// TwinCAT 3 PLC project TcoCognexVision
// Title: TcoCognexVision
// Company: Vortex.Library
// ProjectVersion: 0.6.0.913
// ProgramVersion: 3.1.4023.0
// libraries:
//   Tc2_Standard, * (Beckhoff Automation GmbH)
//   Tc2_System, * (Beckhoff Automation GmbH)
//   Tc3_Module, * (Beckhoff Automation GmbH)
//   TcoAbstractions, 0.6.0.913 (Vortex.Library)
//   TcoCore, 0.6.0.913 (Vortex.Library)
//   TcoIo, 0.6.0.913 (Vortex.Library)
//   TcoUtilities, 0.6.0.913 (Vortex.Library)
// project tree:
//   / PlcTask.TcTTO (not stored)
//   POUs/TcoDataman/v_5_x_x/IO/ TcoDatamanAcquisitionControl_v_5_x_x.TcDUT (not stored), TcoDatamanAcquisitionStatus_v_5_x_x.TcDUT (not stored), TcoDatamanIO_v_5_x_x.TcDUT (not stored), TcoDatamanResultData_v_5_x_x.TcDUT (not stored), TcoDatamanResultsControl_v_5_x_x.TcDUT (not stored), TcoDatamanResultsStatus_v_5_x_x.TcDUT (not stored), TcoDatamanSoftEventControl_v_5_x_x.TcDUT (not stored), TcoDatamanUserData_v_5_x_x.TcDUT (not stored)
//   POUs/TcoDataman/v_5_x_x/Structs/ eDatamanResultDataSize_v_5_x_x.TcDUT (not stored), eDatamanUserDataSize_v_5_x_x.TcDUT (not stored), TcoDatamanConfig_v_5_x_x.TcDUT, TcoDatamanResults_v_5_x_x.TcDUT (not stored), TcoDatamanSignalStates_v_5_x_x.TcDUT (not stored), TcoDatamanStatus_v_5_x_x.TcDUT, TcoDatamanUser_v_5_x_x.TcDUT (not stored)
//   POUs/TcoDataman/v_5_x_x/Tasks/ TcoDatamanClearResultData_v_5_x_x.TcPOU, TcoDatamanRead_v_5_x_x.TcPOU
//   POUs/TcoDataman/v_5_x_x/ TcoDataman_v_5_x_x.TcPOU
//   POUs/TcoDesigner/Structs/ eTcoDesignerTriggerType.TcDUT (not stored), TcoDesignerConfig_v_2_x_x.TcDUT, TcoDesignerData_2_x_x.TcDUT (not stored), TcoDesignerRootContainer.TcPOU (not stored), TcoDesignerStatus_v_2_x_x.TcDUT (not stored), TcoDesignerGenericResults_v_2_x_x.TcDUT (not stored), TcoDesignerPcToPlc_v_2_x_x.TcDUT (not stored), TcoDesignerPlcToPc_v_2_x_x.TcDUT (not stored)
//   POUs/TcoDesigner/Tasks/ TcoDesignerTrigger_v_2_x_x.TcPOU, TcoDesignerClearInspectionResults_v_2_x_x.TcPOU
//   POUs/TcoDesigner/ TcoDesigner_v_2_x_x.TcPOU (not stored)
//   POUs/TcoInsight/v_5_x_x/IO/ TcoInsightAcquisitionControl_v_5_x_x.TcDUT (not stored), TcoInsightAcquisitionStatus_v_5_x_x.TcDUT (not stored), TcoInsightIO_v_5_x_x.TcDUT (not stored), TcoInsightResultData_v_5_x_x.TcDUT (not stored), TcoInsightInspectionControl_v_5_x_x.TcDUT (not stored), TcoInsightInspectionStatus_v_5_x_x.TcDUT (not stored), TcoInsightSoftEventControl_v_5_x_x.TcDUT (not stored), TcoInsightCommandControl_v_5_x_x.TcDUT (not stored), TcoInsightUserData_v_5_x_x.TcDUT (not stored)
//   POUs/TcoInsight/v_5_x_x/Structs/ eTcoInsightResultDataSize_v_5_x_x.TcDUT (not stored), eTcoInsightUserDataSize_v_5_x_x.TcDUT (not stored), TcoInsightConfig_v_5_x_x.TcDUT, TcoInsightResults_v_5_x_x.TcDUT (not stored), TcoInsightSignalStates_v_5_x_x.TcDUT (not stored), TcoInsightStatus_v_5_x_x.TcDUT (not stored), TcoInsightUser_v_5_x_x.TcDUT (not stored)
//   POUs/TcoInsight/v_5_x_x/Tasks/ TcoInsightSetUserData_v_5_x_x.TcPOU, TcoInsightClearUserData_v_5_x_x.TcPOU, TcoInsightTrigger_v_5_x_x.TcPOU, TcoInsightChangeJobByName_v_5_x_x.TcPOU, TcoInsightChangeJobByNumber_v_5_x_x.TcPOU, TcoInsightClearInspectionResults_v_5_x_x.TcPOU, TcoInsightSoftEvent_v_5_x_x.TcPOU
//   POUs/TcoInsight/v_5_x_x/ TcoInsight_v_5_x_x.TcPOU
//   POUs/ TcoVisionParams.TcGVL (not stored)

// ---- POUs/TcoDataman/v_5_x_x/Structs/TcoDatamanConfig_v_5_x_x.TcDUT
TYPE
    TcoDatamanConfig_v_5_x_x :
    STRUCT
        ResultDataSize : eDatamanResultDataSize_v_5_x_x := eDatamanResultDataSize_v_5_x_x.RESULT_DATA_64B;
        UserDataSize : eDatamanUserDataSize_v_5_x_x := eDatamanUserDataSize_v_5_x_x.USER_DATA_64B;
        DataFormat : eTcoDataFormat := TcoUtilities.eTcoDataFormat.BigEndian;
		{attribute addProperty Name "<#Continuous Reading (Hand-held reader)#>"}
        ContinuousReading : BOOL := FALSE;
		UpdateStatesPermanently : BOOL := TRUE;
        InfoTime : TIME := T#2S;
        ErrorTime : TIME := T#5S;
		ShowUserData : BOOL := FALSE;
		ShowResultsData : BOOL := FALSE;
    END_STRUCT
END_TYPE

// ---- POUs/TcoDataman/v_5_x_x/Structs/TcoDatamanStatus_v_5_x_x.TcDUT
TYPE TcoDatamanStatus_v_5_x_x :
STRUCT
	ActionDescription : STRING(100);
	ResultString:STRING(254);
	
	SignalStatus : TcoDatamanSignalStates_v_5_x_x;
END_STRUCT
END_TYPE

// ---- POUs/TcoDesigner/Structs/TcoDesignerConfig_v_2_x_x.TcDUT
TYPE
    TcoDesignerConfig_v_2_x_x :
    STRUCT
   
      
		TriggerTimemout : TIME := T#15S;
		ConnectionTimemout : TIME := T#10S;
        InfoTime : TIME := T#2S;
        ErrorTime : TIME := T#0S;
    END_STRUCT
END_TYPE

// ---- POUs/TcoInsight/v_5_x_x/Structs/TcoInsightConfig_v_5_x_x.TcDUT
TYPE
    TcoInsightConfig_v_5_x_x :
    STRUCT
        ResultDataSize : eTcoInsightResultDataSize_v_5_x_x := eTcoInsightResultDataSize_v_5_x_x.RESULT_DATA_64B;
        UserDataSize : eTcoInsightUserDataSize_v_5_x_x := eTcoInsightUserDataSize_v_5_x_x.USER_DATA_64B;
        DataFormat : eTcoDataFormat := TcoUtilities.eTcoDataFormat.BigEndian;
		UpdateStatesPermanently : BOOL := FALSE;
        MaxJobNumber : UINT := 999;
        InfoTime : TIME := T#2S;
        ErrorTime : TIME := T#0S;
		ShowUserData : BOOL := FALSE;
		ShowResultsData : BOOL := FALSE;

    //	ServiceJobNumber		:	UINT;
    //	ServiceJobName			:	STRING;
    //	ServiceSoftEventNumber	:	UINT;
    END_STRUCT
END_TYPE

// ---- POUs/TcoDataman/v_5_x_x/Tasks/TcoDatamanClearResultData_v_5_x_x.TcPOU
FUNCTION_BLOCK TcoDatamanClearResultData_v_5_x_x EXTENDS TcoCore.TcoTask
VAR_IN_OUT
	inoIoData : TcoDatamanIO_v_5_x_x;
    inoConfig : TcoDatamanConfig_v_5_x_x;
	inoStatus : TcoDatamanStatus_v_5_x_x;	
	inoResults : TcoDatamanResults_v_5_x_x;
END_VAR
VAR
    {attribute 'hide'} 
	_progress : INT := 0;
    {attribute 'hide'} 
	_infoTimer :  TON;
    {attribute 'hide'} 
	_errorTimer :  TON;
    {attribute 'hide'} 
	_varInfo : __SYSTEM.VAR_INFO;
    {attribute 'hide'} 
	_sb : TcoCore.StringBuilder;
END_VAR

IF Execute() THEN
	IF _progress = 0 THEN
		IF NOT __ISVALIDREF(inoIoData) THEN
			_varInfo :=__VARINFO(inoIoData);
			Messenger.Programming(_sb.Clear().Append('<#Invalid reference: #>').Append(_varInfo.Symbol).ToString()).Pin();
		ELSIF NOT __ISVALIDREF(inoConfig) THEN                                                  
			_varInfo :=__VARINFO(inoConfig);                                                    
			Messenger.Programming(_sb.Clear().Append('<#Invalid reference: #>').Append(_varInfo.Symbol).ToString()).Pin();
		ELSIF NOT __ISVALIDREF(inoStatus) THEN                                                  
			_varInfo :=__VARINFO(inoStatus);                                                    
			Messenger.Programming(_sb.Clear().Append('<#Invalid reference: #>').Append(_varInfo.Symbol).ToString()).Pin();
		ELSIF NOT __ISVALIDREF(inoResults) THEN                                              
			_varInfo :=__VARINFO(inoResults);                                                
			Messenger.Programming(_sb.Clear().Append('<#Invalid reference: #>').Append(_varInfo.Symbol).ToString()).Pin();
		ELSE
			_progress := _progress + 1;
		END_IF
	END_IF
	
	IF _progress = 1 THEN
		THIS^.inoStatus.ActionDescription := '<#Clearing of the result data running.#>'; 
		CallTimers(FALSE);
		_progress := _progress + 1;
	END_IF
	
	IF _progress = 2 THEN
		THIS^.inoIoData.AcquisitionControl.TriggerEnable := FALSE;
		THIS^.inoIoData.AcquisitionControl.Trigger := FALSE;
		THIS^.inoIoData.ResultsControl.ResultsAcknowledge := TRUE;
		THIS^.Messenger.OnCondition(_infoTimer.Q).Warning('<#Waiting for the result data cleared!#>').Pin();
		THIS^.inoResults.Length := 0; 
		IF Tc2_System.MEMSET(destAddr:= ADR(THIS^.inoResults.Data) , fillByte:= 0 , n:= SIZEOF(THIS^.inoResults.Data)) >0 THEN
			CallTimers(FALSE);
			_progress := _progress + 1;
		END_IF
	END_IF
	
	IF _progress = 3 THEN
		THIS^.Messenger.OnCondition(_infoTimer.Q).Warning('<#Waiting for the signal ResultsAvailable to be reseted!#>').Pin(); 
		IF NOT THIS^.inoIoData.ResultsStatus.ResultsAvailable THEN
			CallTimers(FALSE);
			_progress := _progress + 1;
		END_IF
	END_IF
	
	IF _progress = 4 THEN
		THIS^.inoIoData.ResultsControl.ResultsAcknowledge := FALSE;
		THIS^.DoneWhen(TRUE);
		CallTimers(FALSE);
		_progress := 0;
	END_IF
	
	CallTimers(TRUE);
	
	THIS^.ThrowWhen(_errorTimer.Q);
END_IF

METHOD CallTimers
VAR_INPUT
	inValue : BOOL;
END_VAR
IF  __ISVALIDREF(inoConfig) AND THIS^.inoConfig.ErrorTime <> T#0S OR NOT inValue THEN  
_errorTimer(IN := inValue, PT := THIS^.inoConfig.ErrorTime);
END_IF;
IF  __ISVALIDREF(inoConfig) AND THIS^.inoConfig.InfoTime <>T#0S OR NOT inValue THEN  
_infoTimer(IN := inValue, PT := THIS^.inoConfig.InfoTime);
END_IF;
END_METHOD

{attribute 'hide'}
METHOD PUBLIC FB_init : BOOL
VAR_INPUT
	bInitRetains : BOOL; // if TRUE, the retain variables are initialized (warm start / cold start)
	bInCopyCode : BOOL;  // if TRUE, the instance afterwards gets moved into the copy code (online change)
	ParentObject : ITcoObject;
END_VAR
END_METHOD

(*~
	<docu>
		<summary>
			Executes when task is aborted.
		</summary>			
	</docu>	
~*)
METHOD PROTECTED OnAbort
THIS^.inoStatus.ActionDescription := '<#Clearing of the result data was aborted, while not yet completed!#>';
END_METHOD

(*~
	<docu>
		<summary>
			Executes when task reaches the ```Done``` state .
		</summary>			
	</docu>	
~*)
METHOD PROTECTED OnDone
THIS^.inoStatus.ActionDescription := '<#Clearing of the result data was completed successfully.#>';
END_METHOD

(*~
	<docu>
		<summary>
			Executes when task reaches the ```Error``` state.
			<para>
				Do not confuse with <see cref="PlcDocu.TcoCore.TcoTask.WhileError()"/>, that is called cyclically until '''Error''' state is left.
			</para>
		</summary>			
	</docu>	
~*)
METHOD PROTECTED OnError
THIS^.inoStatus.ActionDescription := '<#Clearing of the result data finished with error.#>';
END_METHOD

METHOD PROTECTED OnStart
THIS^.inoStatus.ActionDescription := '<#Clearing of the result data started.#>';
END_METHOD

(*~
	<docu>
		<summary>
			Restores this instance to the Ready state. Can be called explicitly or from within one of the restore mechanisms.
			<para>
				See also <see cref="PlcDocu.TcoCore.TcoTask.AutoRestorable()"/>
			</para>
		</summary>			
	</docu>	
~*)
METHOD Restore : ITcoRestorable
SUPER^.Restore();
_progress := 0;
CallTimers(FALSE);
Messenger.UnPin();
END_METHOD

END_FUNCTION_BLOCK

// ---- POUs/TcoDataman/v_5_x_x/Tasks/TcoDatamanRead_v_5_x_x.TcPOU
FUNCTION_BLOCK TcoDatamanRead_v_5_x_x EXTENDS TcoCore.TcoTask
VAR_IN_OUT
	inoIoData 	: TcoDatamanIO_v_5_x_x;
    inoConfig 	: TcoDatamanConfig_v_5_x_x;
	inoStatus 	: TcoDatamanStatus_v_5_x_x;	
	inoResults 	: TcoDatamanResults_v_5_x_x;
END_VAR
VAR
    {attribute 'hide'} 
	_progress : INT := 0;
    {attribute 'hide'} 
	_infoTimer :  TON;
    {attribute 'hide'} 
	_errorTimer :  TON;
    {attribute 'hide'} 
	_varInfo : __SYSTEM.VAR_INFO;
    {attribute 'hide'} 
	_sb : TcoCore.StringBuilder;
END_VAR

IF Execute() THEN
	IF _progress = 0 THEN
		IF NOT __ISVALIDREF(inoIoData) THEN
			_varInfo :=__VARINFO(inoIoData);
			Messenger.Programming(_sb.Clear().Append('<#Invalid reference: #>').Append(_varInfo.Symbol).ToString()).Pin();
		ELSIF NOT __ISVALIDREF(inoConfig) THEN                                                  
			_varInfo :=__VARINFO(inoConfig);                                                    
			Messenger.Programming(_sb.Clear().Append('<#Invalid reference: #>').Append(_varInfo.Symbol).ToString()).Pin();
		ELSIF NOT __ISVALIDREF(inoStatus) THEN                                                  
			_varInfo :=__VARINFO(inoStatus);                                                    
			Messenger.Programming(_sb.Clear().Append('<#Invalid reference: #>').Append(_varInfo.Symbol).ToString()).Pin();
		ELSIF NOT __ISVALIDREF(inoResults) THEN                                              
			_varInfo :=__VARINFO(inoResults);                                                
			Messenger.Programming(_sb.Clear().Append('<#Invalid reference: #>').Append(_varInfo.Symbol).ToString()).Pin();
		ELSE
			_progress := _progress + 1;
		END_IF
	END_IF
	
	IF _progress = 1 THEN
		THIS^.inoStatus.ActionDescription := '<#Reading running.#>'; 
		CallTimers(FALSE);
		_progress := _progress + 1;
	END_IF
	
	IF _progress = 2 THEN
		THIS^.inoIoData.AcquisitionControl.TriggerEnable := TRUE;
		THIS^.inoIoData.AcquisitionControl.Trigger := FALSE;
		THIS^.inoIoData.ResultsControl.EnableResultBuffering := FALSE;
		THIS^.inoIoData.ResultsControl.ResultsAcknowledge := THIS^.inoIoData.ResultsStatus.ResultsAvailable;
		THIS^.Messenger.OnCondition(_infoTimer.Q).Warning('<#Waiting for the signal ResultsAvailable to be reseted!#>').Pin(); 
		IF NOT THIS^.inoIoData.ResultsStatus.ResultsAvailable THEN
			CallTimers(FALSE);
			_progress := _progress + 1;
		END_IF
	END_IF
	
	IF _progress = 3 THEN
		THIS^.Messenger.OnCondition(_infoTimer.Q).Warning('<#Waiting for the signal TriggerReady to be set!#>').Pin(); 
		IF THIS^.inoIoData.AcquisitionStatus.TriggerReady THEN
			CallTimers(FALSE);
			_progress := _progress + 1;
		END_IF
	END_IF
	
	IF _progress = 4 THEN
		THIS^.inoIoData.AcquisitionControl.Trigger := TRUE;
		THIS^.Messenger.OnCondition(_infoTimer.Q).Warning('<#Waiting for the signal TriggerAcknowledge to be set!#>').Pin(); 
		IF THIS^.inoIoData.AcquisitionStatus.TriggerAcknowledge THEN
			CallTimers(FALSE);
			_progress := _progress + 1;
		END_IF
	END_IF
	
	IF _progress = 5 THEN
		THIS^.Messenger.OnCondition(_infoTimer.Q).Warning('<#Waiting for the signal ResultsAvailable to be set!#>').Pin(); 
		IF THIS^.inoIoData.ResultsStatus.ResultsAvailable THEN
			CallTimers(FALSE);
			_progress := _progress + 1;
		END_IF
	END_IF
	
	IF _progress = 6 THEN
		THIS^.inoResults.Length := THIS^.inoIoData.ResultData.ResultLength;
		THIS^.Messenger.OnCondition(_infoTimer.Q).Warning('<#Waiting for the ResultData copied!#>').Pin(); 
		IF  THIS^.inoIoData.ResultData.ResultCode.0=1 THEN // read successfull
			IF Tc2_System.MEMCPY(srcAddr := ADR(THIS^.inoIoData.ResultData.ResultData) , destAddr:= ADR(THIS^.inoResults.Data) ,  n:= THIS^.inoResults.Length) > 0 AND 
				Tc2_System.MEMSET(destAddr:= ADR(THIS^.inoResults.Data) + THIS^.inoResults.Length, fillByte:= 0 , n:= SIZEOF(THIS^.inoResults.Data) - THIS^.inoResults.Length)>0 THEN
				CallTimers(FALSE);
				_progress := _progress + 1;
			END_IF;
		ELSIF THIS^.inoIoData.ResultData.ResultCode.0=0  THEN  // read not successfull
			Tc2_System.MEMSET(destAddr:= ADR(THIS^.inoIoData) , fillByte:= 0 , n:= SIZEOF(THIS^.inoIoData));
			CallTimers(FALSE);
			_progress := _progress + 1;
		
		END_IF
	END_IF
	
	IF _progress = 7 THEN
		THIS^.inoIoData.AcquisitionControl.Trigger := FALSE;
		THIS^.inoIoData.ResultsControl.EnableResultBuffering := FALSE;
		THIS^.inoIoData.ResultsControl.ResultsAcknowledge := TRUE;
		//THIS^.ThrowWhen(THIS^.inoIoData.ResultData.ResultCode=0 OR THIS^.inoIoData.ResultData.ResultLength=0);
		THIS^.DoneWhen(TRUE);
		_progress := 0;
	END_IF
	THIS^.ThrowWhen(THIS^.inoIoData.AcquisitionStatus.MissedAcquisition );
	THIS^.ThrowWhen(THIS^.inoIoData.ResultsStatus.ErrorDetected);

	CallTimers(TRUE);
	
	THIS^.ThrowWhen(_errorTimer.Q);
	
END_IF

METHOD CallTimers
VAR_INPUT
	inValue : BOOL;
END_VAR
IF  __ISVALIDREF(inoConfig) AND THIS^.inoConfig.ErrorTime <> T#0S OR NOT inValue THEN  
_errorTimer(IN := inValue, PT := THIS^.inoConfig.ErrorTime);
END_IF;
IF  __ISVALIDREF(inoConfig) AND THIS^.inoConfig.InfoTime <>T#0S OR NOT inValue THEN  
_infoTimer(IN := inValue, PT := THIS^.inoConfig.InfoTime);
END_IF;
END_METHOD

{attribute 'hide'}
METHOD PUBLIC FB_init : BOOL
VAR_INPUT
	bInitRetains : BOOL; // if TRUE, the retain variables are initialized (warm start / cold start)
	bInCopyCode : BOOL;  // if TRUE, the instance afterwards gets moved into the copy code (online change)
	ParentObject : ITcoObject;
END_VAR
END_METHOD

(*~
	<docu>
		<summary>
			Executes when task is aborted.
		</summary>			
	</docu>	
~*)
METHOD PROTECTED OnAbort
THIS^.inoStatus.ActionDescription := '<#Reading was aborted, while not yet completed!#>';
END_METHOD

(*~
	<docu>
		<summary>
			Executes when task reaches the ```Done``` state .
		</summary>			
	</docu>	
~*)
METHOD PROTECTED OnDone
THIS^.inoStatus.ActionDescription := '<#Reading was completed successfully.#>';
END_METHOD

(*~
	<docu>
		<summary>
			Executes when task reaches the ```Error``` state.
			<para>
				Do not confuse with <see cref="PlcDocu.TcoCore.TcoTask.WhileError()"/>, that is called cyclically until '''Error''' state is left.
			</para>
		</summary>			
	</docu>	
~*)
METHOD PROTECTED OnError
THIS^.inoStatus.ActionDescription := '<#Reading finished with error.#>';
END_METHOD

METHOD PROTECTED OnStart
THIS^.inoStatus.ActionDescription := '<#Reading started.#>'; 
THIS^.inoStatus.ResultString:='';
END_METHOD

(*~
	<docu>
		<summary>
			Restores this instance to the Ready state. Can be called explicitly or from within one of the restore mechanisms.
			<para>
				See also <see cref="PlcDocu.TcoCore.TcoTask.AutoRestorable()"/>
			</para>
		</summary>			
	</docu>	
~*)
METHOD Restore : ITcoRestorable
SUPER^.Restore();
_progress := 0;
CallTimers(FALSE);
Messenger.UnPin();
END_METHOD

END_FUNCTION_BLOCK

// ---- POUs/TcoDataman/v_5_x_x/TcoDataman_v_5_x_x.TcPOU
FUNCTION_BLOCK TcoDataman_v_5_x_x  EXTENDS TcoIo.TcoPnIoComponent IMPLEMENTS TcoAbstractions.ITcoCodeReader
VAR_IN_OUT
inoIoData : TcoDatamanIO_v_5_x_x;
END_VAR

VAR
	{attribute addProperty Name "<#Config#>"}
    _config : TcoDatamanConfig_v_5_x_x;
	{attribute addProperty Name "<#Status#>"}
	_status : TcoDatamanStatus_v_5_x_x;	
END_VAR

VAR
	{attribute addProperty Name "<#UserData#>"}
	_userData	: TcoDatamanUser_v_5_x_x;
	{attribute addProperty Name "<#Results#>"}
	_results	: TcoDatamanResults_v_5_x_x;
END_VAR

VAR
	{attribute 'hide'}
    _taskEnabled : BOOL;
	{attribute addProperty Name "<#Restore#>"}
    _restoreTask : TcoCore.TcoTask(THIS^);
	{attribute addProperty Name "<#Update signal states#>"}
    _updateSignalStatesTask : TcoCore.TcoTask(THIS^);
	{attribute addProperty Name "<#Clear result data#>"}
    _clearResultDataTask : TcoDatamanClearResultData_v_5_x_x(THIS^);
	{attribute addProperty Name "<#Read#>"}
    _readTask : TcoDatamanRead_v_5_x_x(THIS^);
END_VAR
VAR
    {attribute 'hide'} 
	_varInfo : __SYSTEM.VAR_INFO;
    {attribute 'hide'} 
	_sb : TcoCore.StringBuilder;
END_VAR

IF InvalidReference() THEN
    RETURN;
END_IF

SUPER^(inPnIoBoxState := THIS^.inoIoData.PnIoBoxState,inPnIoBoxDiag := THIS^.inoIoData.PnIoBoxDiag);



IF THIS^._config.ContinuousReading THEN
	ContinuousReading();
END_IF

IF NOT SUPER^.ProfinetReady THEN
	THIS^._status.ActionDescription := '<#Not ready for operation by means of Profinet network!#>';	
END_IF

IF SUPER^.ProfinetReady AND THIS^._status.ActionDescription = '<#Not ready for operation by means of Profinet network!#>' THEN
	THIS^._status.ActionDescription := '<#Ready for operation!#>';	
END_IF

//*************RESTORE********************
_taskEnabled := TRUE;
_restoreTask.Enabled := _taskEnabled;
IF _restoreTask.Execute() THEN
	Restore();
END_IF
//****************************************

//*************UPDATE*********************
IF _config.UpdateStatesPermanently THEN
	UpdateSignalStates();
END_IF;
_taskEnabled := SUPER^.ProfinetReady;
_updateSignalStatesTask.Enabled := _taskEnabled AND NOT _config.UpdateStatesPermanently ;
IF _updateSignalStatesTask.Execute() THEN
	UpdateSignalStates();
END_IF

//****************************************

//*************CLEAR*DATA*****************
_taskEnabled := SUPER^.ProfinetReady AND  NOT _readTask.Busy;
_clearResultDataTask.Enabled := _taskEnabled;
_clearResultDataTask(inoIoData := THIS^.inoIoData,inoConfig := THIS^._config,inoStatus := THIS^._status,inoResults := THIS^._results);
//****************************************

//*************READ***********************
_taskEnabled := SUPER^.ProfinetReady AND NOT _clearResultDataTask.Busy;
_readTask.Enabled :=  _taskEnabled;
_readTask(inoIoData := THIS^.inoIoData,inoConfig := THIS^._config,inoStatus := THIS^._status,inoResults := THIS^._results);

IF NOT _readTask.Busy AND NOT _readTask.Error 
	AND NOT _clearResultDataTask.Busy AND NOT _clearResultDataTask.Error THEN
	_status.ResultString := GetResultAsString(0,_status.SignalStatus.ResultLength);
END_IF;
//****************************************

(*~
	<docu>
		<summary>
			Clears the result data. 		
		</summary>			
	</docu>	
~*)
METHOD ClearResultData : TcoCore.ITcoTaskStatus
ClearResultData := THIS^._clearResultDataTask.Invoke();
END_METHOD

(*~
	<docu>
		<summary>
			Gets the `ClearResultDataTask` task that controls clearing of the results data. 		
		</summary>			
	</docu>	
~*)
PROPERTY ClearResultDataTask : TcoCore.ITcoTaskStatus
GET
ClearResultDataTask := _clearResultDataTask;
END_GET
END_PROPERTY

(*~
	<docu>
		<summary>
			Gets the configuration of the reader. 					
		</summary>			
	</docu>	
~*)
PROPERTY Config : REFERENCE TO TcoDatamanConfig_v_5_x_x
GET
Config REF= _config;
END_GET
END_PROPERTY

METHOD INTERNAL ContinuousReading
IF THIS^.inoIoData.ResultsStatus.ResultsAvailable AND NOT THIS^.inoIoData.ResultsControl.ResultsAcknowledge AND THIS^.inoIoData.ResultData.ResultCode>0 AND  THIS^.inoIoData.ResultData.ResultLength>0 THEN
	THIS^._results.Length := THIS^.inoIoData.ResultData.ResultLength;
	Tc2_System.MEMCPY(srcAddr := ADR(THIS^.inoIoData.ResultData.ResultData) , destAddr:= ADR(THIS^._results.Data) ,  n:= THIS^._results.Length);
	Tc2_System.MEMSET(destAddr:= ADR(THIS^._results.Data) + THIS^._results.Length, fillByte:= 0 , n:= SIZEOF(THIS^._results.Data) - THIS^._results.Length);
	THIS^._status.ActionDescription := '<#New data read.#>';
END_IF

THIS^.inoIoData.ResultsControl.ResultsAcknowledge := THIS^.inoIoData.ResultsStatus.ResultsAvailable;
END_METHOD

METHOD FB_init : BOOL
VAR_INPUT
	bInitRetains : BOOL; // if TRUE, the retain variables are initialized (warm start / cold start)
	bInCopyCode : BOOL;  // if TRUE, the instance afterwards gets moved into the copy code (online change)
	ParentObject : ITcoObject;
END_VAR
END_METHOD

METHOD GetResultAsByte : BYTE
VAR_INPUT
    inPosition : UINT;
END_VAR
VAR
	_size : UINT;
END_VAR
_size := SIZEOF(GetResultAsByte);

IF (inPosition +_size) > THIS^._results.Length THEN
	Messenger.Info('<#Index of the ResultData in the method GetResultAsByte exceeds the length of the data received!#>');
	RETURN;
END_IF

IF (inPosition +_size) > THIS^._config.ResultDataSize THEN
	Messenger.Warning('<#Index of the ResultData in the method GetResultAsByte exceeds the size hardware structure mapped!#>');
	RETURN;
END_IF

IF (inPosition +_size) > TcoVisionParams.MAX_BYTE_ARRAY THEN
	Messenger.Programming('<#Index of the ResultData in the method GetResultAsByte exceeds the defined size!#>');
	RETURN;
END_IF

GetResultAsByte := THIS^._results.Data[inPosition];
END_METHOD

METHOD GetResultAsDint : DINT
VAR_INPUT
    inPosition : UINT;
END_VAR
VAR
	_index : UINT;
	_size : UINT;
END_VAR
_size := SIZEOF(GetResultAsDint);

IF (inPosition +_size) > THIS^._results.Length THEN
	Messenger.Info('<#Index of the ResultData in the method GetResultAsDint exceeds the length of the data received!#>');
	RETURN;
END_IF

IF (inPosition +_size) > THIS^._config.ResultDataSize THEN
	Messenger.Warning('<#Index of the ResultData in the method GetResultAsDint exceeds the size hardware structure mapped!#>');
	RETURN;
END_IF

IF (inPosition +_size) > TcoVisionParams.MAX_BYTE_ARRAY THEN
	Messenger.Programming('<#Index of the ResultData in the method GetResultAsDint exceeds the defined size!#>');
	RETURN;
END_IF

GetResultAsDint := TcoUtilities.TcoBytesToDint(THIS^._config.DataFormat,	THIS^._results.Data[inPosition],
															THIS^._results.Data[inPosition+1],
															THIS^._results.Data[inPosition+2],
															THIS^._results.Data[inPosition+3]);
END_METHOD

METHOD GetResultAsReal : REAL
VAR_INPUT
    inPosition : UINT;
END_VAR
VAR
	_index : UINT;
	_size : UINT;
END_VAR
_size := SIZEOF(GetResultAsReal);

IF (inPosition +_size) > THIS^._results.Length THEN
	Messenger.Info('<#Index of the ResultData in the method GetResultAsReal exceeds the length of the data received!#>');
	RETURN;
END_IF

IF (inPosition +_size) > THIS^._config.ResultDataSize THEN
	Messenger.Warning('<#Index of the ResultData in the method GetResultAsReal exceeds the size hardware structure mapped!#>');
	RETURN;
END_IF

IF (inPosition +_size) > TcoVisionParams.MAX_BYTE_ARRAY THEN
	Messenger.Programming('<#Index of the ResultData in the method GetResultAsReal exceeds the defined size!#>');
	RETURN;
END_IF

GetResultAsReal := TcoUtilities.TcoBytesToReal(THIS^._config.DataFormat,	THIS^._results.Data[inPosition],
															THIS^._results.Data[inPosition+1],
															THIS^._results.Data[inPosition+2],
															THIS^._results.Data[inPosition+3]);
END_METHOD

METHOD GetResultAsString : STRING(254)
VAR_INPUT
    inPosition : UINT;
	inLength : UINT;
END_VAR
VAR
	_index : UINT;
	_bufferSize : UINT; 
	_resultString : STRING;
END_VAR

IF (inPosition +inLength) > THIS^._results.Length THEN
	Messenger.Info('<#Index of the ResultData in the method GetResultAsString exceeds the length of the data received!#>');
	RETURN;
END_IF

IF (inPosition +inLength) > THIS^._config.ResultDataSize THEN
	Messenger.Warning('<#Index of the ResultData in the method GetResultAsString exceeds the size hardware structure mapped!#>');
	RETURN;
END_IF

IF (inPosition +inLength) > TcoVisionParams.MAX_BYTE_ARRAY THEN
	Messenger.Programming('<#Index of the ResultData in the method GetResultAsString exceeds the defined size!#>');
	RETURN;
END_IF

_resultString:='';

IF (inLength>0) THEN 
	FOR	_index := 0 TO inLength-1 BY 1 DO	
		IF(THIS^._results.Data[inPosition + _index] <> 0) THEN
			_resultString := CONCAT(_resultString, F_ToCHR(THIS^._results.Data[inPosition + _index]));
		ELSE
			EXIT;	
		END_IF		
	END_FOR;
END_IF

GetResultAsString := _resultString;
END_METHOD

METHOD INTERNAL InvalidReference : BOOL
InvalidReference := FALSE;
IF NOT __ISVALIDREF(inoIoData) THEN
	_varInfo :=__VARINFO(inoIoData);
	Messenger.Error(_sb.Clear().Append('<#Invalid reference: #>').Append(_varInfo.Symbol).ToString());
    InvalidReference := TRUE;
END_IF
END_METHOD

(*~
	<docu>
		<summary>
			Gets the last results data. 		
		</summary>			
	</docu>	
~*)
PROPERTY LastResultData : TcoDatamanResults_v_5_x_x
GET
LastResultData := THIS^._results;
END_GET
END_PROPERTY

(*~
	<docu>
		<summary>
			Triggers the reading sequence and waits for results. 		
		</summary>			
	</docu>	
~*)
METHOD Read : TcoCore.ITcoTaskStatus
Read := THIS^._readTask.Invoke();
END_METHOD

(*~
	<docu>
		<summary>
			Gets the `ReadTask` task that controls the reading sequence. 		
		</summary>			
	</docu>	
~*)
PROPERTY ReadTask : TcoCore.ITcoTaskStatus
GET
ReadTask := _readTask;
END_GET
END_PROPERTY

(*~
	<docu>
		<summary>
			Restores this instance to the Ready state. Can be called explicitly or from within one of the restore mechanisms.	
		</summary>			
	</docu>	
~*)
METHOD Restore : ITcoRestorable
_updateSignalStatesTask.Restore();
_clearResultDataTask.Restore();
_readTask.Restore();

Tc2_System.MEMSET(destAddr:= ADR(THIS^._results.Data) , fillByte:= 0 , n:= SIZEOF(THIS^._results.Data));

//THIS^.inoIoData.AcquisitionControl.TriggerEnable := FALSE;
//THIS^.inoIoData.AcquisitionControl.Trigger := FALSE;

THIS^._results.Code := 0;
THIS^._results.Extended := 0;
THIS^._results.Id := 0;
THIS^._results.Length := 0;
	
IF InvalidReference() THEN
    RETURN;
END_IF

Tc2_System.MEMSET(destAddr:= ADR(THIS^.inoIoData) , fillByte:= 0 , n:= SIZEOF(THIS^.inoIoData));


_status.ActionDescription := '<#Restore executed!#>';
_restoreTask.Restore();
END_METHOD

(*~
	<docu>
		<summary>
		    Custom service (manual, maintenance) logic.
			This method must be implemented in derived class.
		</summary>			
	</docu>	
~*)
METHOD PROTECTED ServiceMode
END_METHOD

(*~
	<docu>
		<summary>
			Gets the status of the reader. 					
		</summary>			
	</docu>	
~*)
PROPERTY Status : REFERENCE TO TcoDatamanStatus_v_5_x_x
GET
Status REF= _status;
END_GET
END_PROPERTY

METHOD INTERNAL UpdateSignalStates
_status.SignalStatus.TriggerEnable 			:=	inoIoData.AcquisitionControl.TriggerEnable; 
_status.SignalStatus.Trigger				:=	inoIoData.AcquisitionControl.Trigger; 

_status.SignalStatus.EnableResultBuffering	:=	inoIoData.ResultsControl.EnableResultBuffering;
_status.SignalStatus.ResultsAcknowledge		:=	inoIoData.ResultsControl.ResultsAcknowledge;

_status.SignalStatus.TriggerReady 			:= 	inoIoData.AcquisitionStatus.TriggerReady;
_status.SignalStatus.TriggerAcknowledge 	:= 	inoIoData.AcquisitionStatus.TriggerAcknowledge;
_status.SignalStatus.Acquiring 				:= 	inoIoData.AcquisitionStatus.Acquiring;
_status.SignalStatus.MissedAcquisition 		:= 	inoIoData.AcquisitionStatus.MissedAcquisition;
_status.SignalStatus.TriggerID 				:= 	inoIoData.AcquisitionStatus.TriggerID;

_status.SignalStatus.Decoding 				:= 	inoIoData.ResultsStatus.Decoding;
_status.SignalStatus.DecodeComplete 		:= 	inoIoData.ResultsStatus.DecodeComplete;
_status.SignalStatus.ResultsBufferOverrun 	:= 	inoIoData.ResultsStatus.ResultsBufferOverrun;
_status.SignalStatus.ResultsAvailable 		:= 	inoIoData.ResultsStatus.ResultsAvailable;
_status.SignalStatus.ErrorDetected 			:= 	inoIoData.ResultsStatus.ErrorDetected;

_status.SignalStatus.ResultID 				:= 	inoIoData.ResultData.ResultID;
_status.SignalStatus.ResultCode  			:= 	inoIoData.ResultData.ResultCode;
_status.SignalStatus.ResultExtended  		:= 	inoIoData.ResultData.ResultExtended;
_status.SignalStatus.ResultLength  			:= 	inoIoData.ResultData.ResultLength;

_updateSignalStatesTask.DoneWhen(TRUE);
END_METHOD

END_FUNCTION_BLOCK

// ---- POUs/TcoDesigner/Tasks/TcoDesignerTrigger_v_2_x_x.TcPOU
FUNCTION_BLOCK TcoDesignerTrigger_v_2_x_x EXTENDS TcoCore.TcoTask
VAR_INPUT
	inTriggerType:eTcoDesignerTriggerType;
	refClearResultsTask: REFERENCE TO TcoDesignerClearInspectionResults_v_2_x_x;
END_VAR 

VAR
	_clearResultsTask: REFERENCE TO TcoDesignerClearInspectionResults_v_2_x_x;
END_VAR
VAR_IN_OUT
	inoIoData	: TcoDesignerData_2_x_x;
    inoConfig	: TcoDesignerConfig_v_2_x_x;
	inoStatus	: TcoDesignerStatus_v_2_x_x;	
	//inoResults	: TcoInsightResults_v_5_x_x;
END_VAR
VAR
   
	_progress : INT := 0;
    {attribute 'hide'} 
	_infoTimer :  TON;
    {attribute 'hide'} 
	_errorTimer :  TON;
    {attribute 'hide'} 
	_varInfo : __SYSTEM.VAR_INFO;
    {attribute 'hide'} 
	_sb : TcoCore.StringBuilder;
  
END_VAR

IF NOT __ISVALIDREF(refClearResultsTask)  THEN
    Messenger.Post('<#Invalid reference ClearResultsTask>', TcoCore.eMessageCategory.ProgrammingError);
    RETURN;
END_IF
_clearResultsTask REF= refClearResultsTask;

IF Execute() THEN
	IF _progress = 0 THEN
		IF NOT __ISVALIDREF(inoIoData) THEN
			_varInfo :=__VARINFO(inoIoData);
			Messenger.Programming(_sb.Clear().Append('<#Invalid reference: #>').Append(_varInfo.Symbol).ToString()).Pin();
		ELSIF NOT __ISVALIDREF(inoConfig) THEN                                                  
			_varInfo :=__VARINFO(inoConfig);                                                    
			Messenger.Programming(_sb.Clear().Append('<#Invalid reference: #>').Append(_varInfo.Symbol).ToString()).Pin();
		ELSIF NOT __ISVALIDREF(inoStatus) THEN                                                  
			_varInfo :=__VARINFO(inoStatus);                                                    
			Messenger.Programming(_sb.Clear().Append('<#Invalid reference: #>').Append(_varInfo.Symbol).ToString()).Pin();

		ELSIF inTriggerType = eTcoDesignerTriggerType.TriggerWithTimeout 
			AND inoConfig.ErrorTime < inoConfig.TriggerTimemout  AND inoConfig.ErrorTime <>T#0S THEN
				Messenger.Error(_sb.Clear().Append('<#Error time is lower than timeout. Please check config!#>').ToString()).Pin();

		ELSE
			_progress := _progress + 1;
			CallTimers(FALSE);

		END_IF
	END_IF
	
		
	IF _progress = 1 THEN
		IF inTriggerType = eTcoDesignerTriggerType.TriggerFast THEN
			_progress := _progress + 1;
		ELSIF inTriggerType = eTcoDesignerTriggerType.TriggerWithTimeout THEN
			inoIoData.PlcToPc.Timeout:=TIME_TO_UINT( inoConfig.TriggerTimemout);
			IF _clearResultsTask.Invoke().Done THEN
				_progress := _progress + 1;
			END_IF;
		ELSIF _clearResultsTask.Invoke().Done THEN
			_progress := _progress + 1;
		END_IF

	END_IF;
	
	IF _progress = 2 THEN
		THIS^.Messenger.OnCondition(_infoTimer.Q).Warning('<#Waiting for the Online signal!#>'); 
		IF THIS^.inoIoData.PcToPlc.SystemOnline THEN
			CallTimers(FALSE);
			_progress := _progress + 1;
		END_IF
	END_IF
	

	IF _progress = 3 THEN
		THIS^.Messenger.OnCondition(_infoTimer.Q).Info('<#Trigger!#>'); 
		THIS^.inoIoData.PlcToPc.Trigger:=TRUE;
	
		IF NOT THIS^.inoIoData.PcToPlc.InspectionReady  THEN
			THIS^.inoIoData.PlcToPc.Trigger:=FALSE;
			CallTimers(FALSE);
			_progress := _progress + 1;
		END_IF
	END_IF
	
	
	IF _progress=4 THEN	
		Messenger.Info('Waiting for results available');
		IF THIS^.inoIoData.PcToPlc.ResultsAvailable  THEN		
			CallTimers(FALSE);
			_progress := _progress + 1;
		END_IF
	END_IF
	
	IF _progress=5 THEN	
		Messenger.Info('Acknovledge results');
		THIS^.inoIoData.PlcToPc.ResultsAck:=TRUE;
		IF NOT THIS^.inoIoData.PcToPlc.ResultsAvailable  THEN
			THIS^.inoIoData.PlcToPc.ResultsAck:=FALSE;
			THIS^.DoneWhen(TRUE);
			
		END_IF
	END_IF
	

	

	CallTimers(TRUE);
	
	THIS^.ThrowWhen(_errorTimer.Q  OR THIS^.inoIoData.PcToPlc.Error 
		OR (inTriggerType = eTcoDesignerTriggerType.TriggerWithTimeout AND THIS^.inoIoData.PcToPlc.TriggerTimeout) );	

END_IF

METHOD CallTimers
VAR_INPUT
	inValue : BOOL;
END_VAR
IF  __ISVALIDREF(inoConfig) AND THIS^.inoConfig.ErrorTime <> T#0S OR NOT inValue THEN  
_errorTimer(IN := inValue, PT := THIS^.inoConfig.ErrorTime);
END_IF;
IF  __ISVALIDREF(inoConfig) AND THIS^.inoConfig.InfoTime <>T#0S OR NOT inValue THEN  
_infoTimer(IN := inValue, PT := THIS^.inoConfig.InfoTime);
END_IF;
END_METHOD

(*~
	<docu>
		<summary>
			Executes when task is aborted.
		</summary>			
	</docu>	
~*)
METHOD PROTECTED OnAbort
THIS^.inoStatus.ActionDescription := '<#Trigger was aborted, while not yet completed!#>';
END_METHOD

(*~
	<docu>
		<summary>
			Executes when task reaches the ```Done``` state .
		</summary>			
	</docu>	
~*)
METHOD PROTECTED OnDone
THIS^.inoStatus.ActionDescription := '<#Trigger was completed successfully.#>'; 
_progress:=0;
END_METHOD

(*~
	<docu>
		<summary>
			Executes when task reaches the ```Error``` state.
			<para>
				Do not confuse with <see cref="PlcDocu.TcoCore.TcoTask.WhileError()"/>, that is called cyclically until '''Error''' state is left.
			</para>
		</summary>			
	</docu>	
~*)
METHOD PROTECTED OnError
THIS^.inoStatus.ActionDescription := '<#Trigger finished with error.#>';
END_METHOD

METHOD PROTECTED OnStart
THIS^.inoStatus.ActionDescription := '<#Trigger started.#>'; 
inoIoData.PlcToPc.Timeout:=0;
END_METHOD

(*~
	<docu>
		<summary>
			Restores this instance to the Ready state. Can be called explicitly or from within one of the restore mechanisms.
			<para>
				See also <see cref="PlcDocu.TcoCore.TcoTask.AutoRestorable()"/>
			</para>
		</summary>			
	</docu>	
~*)
METHOD Restore : ITcoRestorable
SUPER^.Restore();
_progress := 0;
CallTimers(FALSE);
Messenger.UnPin();
END_METHOD

END_FUNCTION_BLOCK

// ---- POUs/TcoDesigner/Tasks/TcoDesignerClearInspectionResults_v_2_x_x.TcPOU
FUNCTION_BLOCK TcoDesignerClearInspectionResults_v_2_x_x EXTENDS TcoCore.TcoTask
VAR_IN_OUT
	inoIoData	: TcoDesignerData_2_x_x;
    inoConfig	: TcoDesignerConfig_v_2_x_x;
	inoStatus	: TcoDesignerStatus_v_2_x_x;	
	//inoResults	: TcoInsightResults_v_5_x_x;
END_VAR
VAR
    {attribute 'hide'} 
	_progress : INT := 0;
    {attribute 'hide'} 
	_infoTimer :  TON;
    {attribute 'hide'} 
	_errorTimer :  TON;
    {attribute 'hide'} 
	_varInfo : __SYSTEM.VAR_INFO;
    {attribute 'hide'} 
	_sb : TcoCore.StringBuilder;
END_VAR

IF Execute() THEN
	IF _progress = 0 THEN
		IF NOT __ISVALIDREF(inoIoData) THEN
			_varInfo :=__VARINFO(inoIoData);
			Messenger.Programming(_sb.Clear().Append('<#Invalid reference: #>').Append(_varInfo.Symbol).ToString()).Pin();
		ELSIF NOT __ISVALIDREF(inoConfig) THEN                                                  
			_varInfo :=__VARINFO(inoConfig);                                                    
			Messenger.Programming(_sb.Clear().Append('<#Invalid reference: #>').Append(_varInfo.Symbol).ToString()).Pin();
		ELSIF NOT __ISVALIDREF(inoStatus) THEN                                                  
			_varInfo :=__VARINFO(inoStatus);                                                    
			Messenger.Programming(_sb.Clear().Append('<#Invalid reference: #>').Append(_varInfo.Symbol).ToString()).Pin();
//		ELSIF NOT __ISVALIDREF(inoResults) THEN                                              
//			_varInfo :=__VARINFO(inoResults);                                                
//			Messenger.Programming(_sb.Clear().Append('<#Invalid reference: #>').Append(_varInfo.Symbol).ToString()).Pin();
		ELSE
			_progress := _progress + 1;
		END_IF
	END_IF
	
	IF _progress = 1 THEN
		CallTimers(FALSE);
		THIS^.inoIoData.PlcToPc.Trigger := FALSE;
		THIS^.inoIoData.PlcToPc.LoadJob := FALSE;
		
		THIS^.inoIoData.PlcToPc.Reset := FALSE;
		THIS^.inoIoData.PlcToPc.ResultsAck := FALSE;

		THIS^.inoIoData.PlcToPc.ClearResults:=FALSE;

		_progress := _progress + 1;
	END_IF
	
	IF _progress = 2 THEN
		THIS^.Messenger.OnCondition(_infoTimer.Q).Info('<#Reset Request!#>'); 
		THIS^.inoIoData.PlcToPc.Reset := TRUE;
		IF THIS^.inoIoData.PcToPlc.InspectionReady
			AND NOT THIS^.inoIoData.PcToPlc.ClearResultsAck
			AND NOT THIS^.inoIoData.PcToPlc.ResultsAvailable 
			AND NOT THIS^.inoIoData.PcToPlc.JobLoadDone THEN
			THIS^.inoIoData.PlcToPc.Reset := FALSE;
			_progress := _progress + 1;
		END_IF
	END_IF
	
	IF _progress = 3 THEN
		THIS^.Messenger.OnCondition(_infoTimer.Q).Warning('<#Waiting for the Online signal!#>'); 
		IF THIS^.inoIoData.PcToPlc.SystemOnline THEN
			CallTimers(FALSE);
			_progress := _progress + 1;
		END_IF
	END_IF
	
	IF _progress = 4 THEN
		THIS^.Messenger.OnCondition(_infoTimer.Q).Info('<#Waiting to Acknowledge results!#>'); 
		THIS^.inoIoData.PlcToPc.ResultsAck:=TRUE;
		IF NOT THIS^.inoIoData.PcToPlc.ResultsAvailable  THEN
			THIS^.inoIoData.PlcToPc.ResultsAck:=FALSE;
			CallTimers(FALSE);
			_progress := _progress + 1;
		END_IF
	END_IF
	
	IF _progress = 5 THEN
		THIS^.Messenger.OnCondition(_infoTimer.Q).Info('<#Waiting to clear old data!#>'); 
		THIS^.inoIoData.PlcToPc.ClearResults:=TRUE;
	
		IF  THIS^.inoIoData.PcToPlc.ClearResultsAck  THEN
			THIS^.inoIoData.PlcToPc.ClearResults:=FALSE;
			CallTimers(FALSE);
			_progress := _progress + 1;
		END_IF
	END_IF
	
	IF _progress = 6 THEN
		THIS^.Messenger.OnCondition(_infoTimer.Q).Info('<#Waiting for Inspection ready!#>'); 
		IF THIS^.inoIoData.PcToPlc.InspectionReady 
			 THEN
			CallTimers(FALSE);
			_progress := _progress + 1;
		END_IF
	END_IF
	
	IF _progress = 7 THEN	
		THIS^.Messenger.OnCondition(_infoTimer.Q).Info('<#Waiting for data were cleared!#>'); 
			IF  NOT THIS^.inoIoData.PcToPlc.ClearResultsAck
			AND NOT THIS^.inoIoData.PcToPlc.InspectionResults.ResultFail
			AND NOT THIS^.inoIoData.PcToPlc.InspectionResults.ResultPass THEN
			CallTimers(FALSE);
			THIS^.DoneWhen(TRUE);
		END_IF
	END_IF
	
	CallTimers(TRUE);
	
		THIS^.ThrowWhen(_errorTimer.Q   OR THIS^.inoIoData.PcToPlc.Error );	
END_IF

METHOD CallTimers
VAR_INPUT
	inValue : BOOL;
END_VAR
IF  __ISVALIDREF(inoConfig) AND THIS^.inoConfig.ErrorTime <> T#0S OR NOT inValue THEN  
_errorTimer(IN := inValue, PT := THIS^.inoConfig.ErrorTime);
END_IF;
IF  __ISVALIDREF(inoConfig) AND THIS^.inoConfig.InfoTime <>T#0S OR NOT inValue THEN  
_infoTimer(IN := inValue, PT := THIS^.inoConfig.InfoTime);
END_IF;
END_METHOD

(*~
	<docu>
		<summary>
			Executes when task is aborted.
		</summary>			
	</docu>	
~*)
METHOD PROTECTED OnAbort
THIS^.inoStatus.ActionDescription := '<#Clearing of the inspection results aborted, while not yet finished.#>';
END_METHOD

(*~
	<docu>
		<summary>
			Executes when task reaches the ```Done``` state .
		</summary>			
	</docu>	
~*)
METHOD PROTECTED OnDone
THIS^.inoStatus.ActionDescription := '<#Clearing of the inspection results was completed succesfully.#>'; 
_progress:=0;
END_METHOD

(*~
	<docu>
		<summary>
			Executes when task reaches the ```Error``` state.
			<para>
				Do not confuse with <see cref="PlcDocu.TcoCore.TcoTask.WhileError()"/>, that is called cyclically until '''Error''' state is left.
			</para>
		</summary>			
	</docu>	
~*)
METHOD PROTECTED OnError
THIS^.inoStatus.ActionDescription := '<#Clearing of the inspection results finished with error.#>';
END_METHOD

METHOD PROTECTED OnStart
THIS^.inoStatus.ActionDescription := '<#Clearing of the inspection results started.#>';
END_METHOD

(*~
	<docu>
		<summary>
			Restores this instance to the Ready state. Can be called explicitly or from within one of the restore mechanisms.
			<para>
				See also <see cref="PlcDocu.TcoCore.TcoTask.AutoRestorable()"/>
			</para>
		</summary>			
	</docu>	
~*)
METHOD Restore : ITcoRestorable
SUPER^.Restore();
_progress := 0;
CallTimers(FALSE);
Messenger.UnPin();
END_METHOD

END_FUNCTION_BLOCK

// ---- POUs/TcoInsight/v_5_x_x/Tasks/TcoInsightSetUserData_v_5_x_x.TcPOU
FUNCTION_BLOCK TcoInsightSetUserData_v_5_x_x EXTENDS TcoCore.TcoTask
VAR_IN_OUT
	inoIoData	: TcoInsightIO_v_5_x_x;
    inoConfig	: TcoInsightConfig_v_5_x_x;
	inoStatus	: TcoInsightStatus_v_5_x_x;	
	inoUserData 	: TcoInsightUser_v_5_x_x;
END_VAR
VAR
    {attribute 'hide'} 
	_progress : INT := 0;
    {attribute 'hide'} 
	_infoTimer :  TON;
    {attribute 'hide'} 
	_errorTimer :  TON;
    {attribute 'hide'} 
	_varInfo : __SYSTEM.VAR_INFO;
    {attribute 'hide'} 
	_sb : TcoCore.StringBuilder;
	   {attribute 'hide'} 
	_size : UINT;
END_VAR

IF Execute() THEN
    IF _progress = 0 THEN
        IF NOT __ISVALIDREF(inoIoData) THEN
            _varInfo := __VARINFO(inoIoData);
            Messenger.Programming(_sb.Clear().Append('<#Invalid reference: #>').Append(_varInfo.Symbol).ToString()).Pin();
        ELSIF NOT __ISVALIDREF(inoConfig) THEN
            _varInfo := __VARINFO(inoConfig);
            Messenger.Programming(_sb.Clear().Append('<#Invalid reference: #>').Append(_varInfo.Symbol).ToString()).Pin();
        ELSIF NOT __ISVALIDREF(inoStatus) THEN
            _varInfo := __VARINFO(inoStatus);
            Messenger.Programming(_sb.Clear().Append('<#Invalid reference: #>').Append(_varInfo.Symbol).ToString()).Pin();
        ELSIF NOT __ISVALIDREF(inoUserData) THEN
            _varInfo := __VARINFO(inoUserData);
            Messenger.Programming(_sb.Clear().Append('<#Invalid reference: #>').Append(_varInfo.Symbol).ToString()).Pin();
        ELSE
            _progress := _progress + 1;
        END_IF
    END_IF

    IF _progress = 1 THEN
        THIS^.inoStatus.ActionDescription := '<#Set user data running.#>';
        CallTimers(FALSE);
        _progress := _progress + 1;
    END_IF

    IF _progress = 2 THEN
        THIS^.inoIoData.InspectionControl.ExecuteCommand := FALSE;
        THIS^.inoIoData.InspectionControl.ClearError := FALSE;
        THIS^.inoIoData.AcquisitionControl.SetOffline := FALSE;

        THIS^.Messenger.OnCondition(_infoTimer.Q).Warning('<#Waiting for the User data to be copied!#>').Pin();

        _size := THIS^.inoConfig.UserDataSize;

        IF Tc2_System.MEMCPY(srcAddr := ADR(THIS^.inoUserData.UserData), destAddr := ADR(THIS^.inoIoData.UserData), n := _size) > 0 AND
            Tc2_System.MEMSET(destAddr := ADR(THIS^.inoIoData.UserData) + _size, fillByte := 0, n := SIZEOF(THIS^.inoIoData.UserData) - _size) > 0
            THEN
            CallTimers(FALSE);
            _progress := _progress + 1;
        END_IF

    END_IF

    IF _progress = 3 THEN
        THIS^.inoIoData.InspectionControl.ExtendedUserDataSet := TRUE;
        Messenger.OnCondition(_infoTimer.Q).Info('<#Waiting for signal User dataset acknowledge#>');

        IF (THIS^.inoIoData.InspectionStatus.ExtendedUserDataSetAcknowledge) THEN
            CallTimers(FALSE);
            _progress := _progress + 1;
        END_IF
    END_IF

    IF _progress = 4 THEN
        THIS^.inoIoData.InspectionControl.ExtendedUserDataSet := FALSE;

        IF (NOT THIS^.inoIoData.InspectionStatus.ExtendedUserDataSetAcknowledge) THEN

            THIS^.DoneWhen(TRUE);
            CallTimers(FALSE);
            _progress := 0;
        END_IF
    END_IF

    CallTimers(TRUE);

    THIS^.ThrowWhen(_errorTimer.Q);
END_IF

METHOD CallTimers
VAR_INPUT
	inValue : BOOL;
END_VAR
IF  __ISVALIDREF(inoConfig) AND THIS^.inoConfig.ErrorTime <> T#0S OR NOT inValue THEN  
_errorTimer(IN := inValue, PT := THIS^.inoConfig.ErrorTime);
END_IF;
IF  __ISVALIDREF(inoConfig) AND THIS^.inoConfig.InfoTime <>T#0S OR NOT inValue THEN  
_infoTimer(IN := inValue, PT := THIS^.inoConfig.InfoTime);
END_IF;
END_METHOD

{attribute 'hide'}
METHOD PUBLIC FB_init : BOOL
VAR_INPUT
	bInitRetains : BOOL; // if TRUE, the retain variables are initialized (warm start / cold start)
	bInCopyCode : BOOL;  // if TRUE, the instance afterwards gets moved into the copy code (online change)
	ParentObject : ITcoObject;
END_VAR
END_METHOD

(*~
	<docu>
		<summary>
			Executes when task is aborted.
		</summary>			
	</docu>	
~*)
METHOD PROTECTED OnAbort
THIS^.inoStatus.ActionDescription := '<#Set user data was aborted, while not yet finished.#>';
END_METHOD

(*~
	<docu>
		<summary>
			Executes when task reaches the ```Done``` state .
		</summary>			
	</docu>	
~*)
METHOD PROTECTED OnDone
THIS^.inoStatus.ActionDescription := '<#Set User data of the inspection  was completed succesfully.#>';
END_METHOD

(*~
	<docu>
		<summary>
			Executes when task reaches the ```Error``` state.
			<para>
				Do not confuse with <see cref="PlcDocu.TcoCore.TcoTask.WhileError()"/>, that is called cyclically until '''Error''' state is left.
			</para>
		</summary>			
	</docu>	
~*)
METHOD PROTECTED OnError
THIS^.inoStatus.ActionDescription := '<#Set user data  finished with error.#>';
END_METHOD

METHOD PROTECTED OnStart
END_METHOD

(*~
	<docu>
		<summary>
			Restores this instance to the Ready state. Can be called explicitly or from within one of the restore mechanisms.
			<para>
				See also <see cref="PlcDocu.TcoCore.TcoTask.AutoRestorable()"/>
			</para>
		</summary>			
	</docu>	
~*)
METHOD Restore : ITcoRestorable
SUPER^.Restore();
_progress := 0;
CallTimers(FALSE);
Messenger.UnPin();
END_METHOD

END_FUNCTION_BLOCK

// ---- POUs/TcoInsight/v_5_x_x/Tasks/TcoInsightClearUserData_v_5_x_x.TcPOU
FUNCTION_BLOCK TcoInsightClearUserData_v_5_x_x EXTENDS TcoCore.TcoTask
VAR_IN_OUT
	inoIoData	: TcoInsightIO_v_5_x_x;
    inoConfig	: TcoInsightConfig_v_5_x_x;
	inoStatus	: TcoInsightStatus_v_5_x_x;	
	inoUserData 	: TcoInsightUser_v_5_x_x;
END_VAR
VAR
    {attribute 'hide'} 
	_progress : INT := 0;
    {attribute 'hide'} 
	_infoTimer :  TON;
    {attribute 'hide'} 
	_errorTimer :  TON;
    {attribute 'hide'} 
	_varInfo : __SYSTEM.VAR_INFO;
    {attribute 'hide'} 
	_sb : TcoCore.StringBuilder;
END_VAR

IF Execute() THEN
    IF _progress = 0 THEN
        IF NOT __ISVALIDREF(inoIoData) THEN
            _varInfo := __VARINFO(inoIoData);
            Messenger.Programming(_sb.Clear().Append('<#Invalid reference: #>').Append(_varInfo.Symbol).ToString()).Pin();
        ELSIF NOT __ISVALIDREF(inoConfig) THEN
            _varInfo := __VARINFO(inoConfig);
            Messenger.Programming(_sb.Clear().Append('<#Invalid reference: #>').Append(_varInfo.Symbol).ToString()).Pin();
        ELSIF NOT __ISVALIDREF(inoStatus) THEN
            _varInfo := __VARINFO(inoStatus);
            Messenger.Programming(_sb.Clear().Append('<#Invalid reference: #>').Append(_varInfo.Symbol).ToString()).Pin();
        ELSIF NOT __ISVALIDREF(inoUserData) THEN
            _varInfo := __VARINFO(inoUserData);
            Messenger.Programming(_sb.Clear().Append('<#Invalid reference: #>').Append(_varInfo.Symbol).ToString()).Pin();
        ELSE
            _progress := _progress + 1;
        END_IF
    END_IF

    IF _progress = 1 THEN
        THIS^.inoStatus.ActionDescription := '<#Set user data running.#>';
        CallTimers(FALSE);
        _progress := _progress + 1;
    END_IF

    IF _progress = 2 THEN
        THIS^.inoIoData.InspectionControl.ExecuteCommand := FALSE;
        THIS^.inoIoData.InspectionControl.ClearError := FALSE;
        THIS^.inoIoData.AcquisitionControl.SetOffline := FALSE;
		IF Tc2_System.MEMSET(destAddr:= ADR(THIS^.inoUserData.UserData) , fillByte:= 0 , n:= SIZEOF(THIS^.inoUserData.UserData)) >0 
			and Tc2_System.MEMSET(destAddr:= ADR(THIS^.inoIoData.UserData) , fillByte:= 0 , n:= SIZEOF(THIS^.inoIoData.UserData)) >0THEN
			CallTimers(FALSE);
			 THIS^.DoneWhen(TRUE);
			 _progress := 0;
		END_IF


    END_IF


    CallTimers(TRUE);

    THIS^.ThrowWhen(_errorTimer.Q);
END_IF

METHOD CallTimers
VAR_INPUT
	inValue : BOOL;
END_VAR
IF  __ISVALIDREF(inoConfig) AND THIS^.inoConfig.ErrorTime <> T#0S OR NOT inValue THEN  
_errorTimer(IN := inValue, PT := THIS^.inoConfig.ErrorTime);
END_IF;
IF  __ISVALIDREF(inoConfig) AND THIS^.inoConfig.InfoTime <>T#0S OR NOT inValue THEN  
_infoTimer(IN := inValue, PT := THIS^.inoConfig.InfoTime);
END_IF;
END_METHOD

{attribute 'hide'}
METHOD PUBLIC FB_init : BOOL
VAR_INPUT
	bInitRetains : BOOL; // if TRUE, the retain variables are initialized (warm start / cold start)
	bInCopyCode : BOOL;  // if TRUE, the instance afterwards gets moved into the copy code (online change)
	ParentObject : ITcoObject;
END_VAR
END_METHOD

(*~
	<docu>
		<summary>
			Executes when task is aborted.
		</summary>			
	</docu>	
~*)
METHOD PROTECTED OnAbort
THIS^.inoStatus.ActionDescription := '<#Clear user data was aborted, while not yet finished.#>';
END_METHOD

(*~
	<docu>
		<summary>
			Executes when task reaches the ```Done``` state .
		</summary>			
	</docu>	
~*)
METHOD PROTECTED OnDone
THIS^.inoStatus.ActionDescription := '<#Userdata of the inspection  was completed succesfully.#>';
END_METHOD

(*~
	<docu>
		<summary>
			Executes when task reaches the ```Error``` state.
			<para>
				Do not confuse with <see cref="PlcDocu.TcoCore.TcoTask.WhileError()"/>, that is called cyclically until '''Error''' state is left.
			</para>
		</summary>			
	</docu>	
~*)
METHOD PROTECTED OnError
THIS^.inoStatus.ActionDescription := '<#User data  finished with error.#>';
END_METHOD

METHOD PROTECTED OnStart
END_METHOD

(*~
	<docu>
		<summary>
			Restores this instance to the Ready state. Can be called explicitly or from within one of the restore mechanisms.
			<para>
				See also <see cref="PlcDocu.TcoCore.TcoTask.AutoRestorable()"/>
			</para>
		</summary>			
	</docu>	
~*)
METHOD Restore : ITcoRestorable
SUPER^.Restore();
_progress := 0;
CallTimers(FALSE);
Messenger.UnPin();
END_METHOD

END_FUNCTION_BLOCK

// ---- POUs/TcoInsight/v_5_x_x/Tasks/TcoInsightTrigger_v_5_x_x.TcPOU
FUNCTION_BLOCK TcoInsightTrigger_v_5_x_x EXTENDS TcoCore.TcoTask
VAR_IN_OUT
	inoIoData	: TcoInsightIO_v_5_x_x;
    inoConfig	: TcoInsightConfig_v_5_x_x;
	inoStatus	: TcoInsightStatus_v_5_x_x;	
	inoResults	: TcoInsightResults_v_5_x_x;
END_VAR
VAR
    {attribute 'hide'} 
	_progress : INT := 0;
    {attribute 'hide'} 
	_infoTimer :  TON;
    {attribute 'hide'} 
	_errorTimer :  TON;
    {attribute 'hide'} 
	_varInfo : __SYSTEM.VAR_INFO;
    {attribute 'hide'} 
	_sb : TcoCore.StringBuilder;
    {attribute 'hide'} 
	_inspectionCompleted : BOOL;
    {attribute 'hide'} 
	_size : UINT;
END_VAR

IF Execute() THEN
	IF _progress = 0 THEN
		IF NOT __ISVALIDREF(inoIoData) THEN
			_varInfo :=__VARINFO(inoIoData);
			Messenger.Programming(_sb.Clear().Append('<#Invalid reference: #>').Append(_varInfo.Symbol).ToString()).Pin();
		ELSIF NOT __ISVALIDREF(inoConfig) THEN                                                  
			_varInfo :=__VARINFO(inoConfig);                                                    
			Messenger.Programming(_sb.Clear().Append('<#Invalid reference: #>').Append(_varInfo.Symbol).ToString()).Pin();
		ELSIF NOT __ISVALIDREF(inoStatus) THEN                                                  
			_varInfo :=__VARINFO(inoStatus);                                                    
			Messenger.Programming(_sb.Clear().Append('<#Invalid reference: #>').Append(_varInfo.Symbol).ToString()).Pin();
		ELSIF NOT __ISVALIDREF(inoResults) THEN                                              
			_varInfo :=__VARINFO(inoResults);                                                
			Messenger.Programming(_sb.Clear().Append('<#Invalid reference: #>').Append(_varInfo.Symbol).ToString()).Pin();
		ELSE
			_progress := _progress + 1;
		END_IF
	END_IF
	
	IF _progress = 1 THEN
		THIS^.inoStatus.ActionDescription := '<#Trigger running.#>'; 
		CallTimers(FALSE);
		THIS^.inoIoData.AcquisitionControl.AcquisitionTriggerEnable := TRUE;
		THIS^.inoIoData.AcquisitionControl.AcquisitionTrigger := FALSE;
		THIS^.inoIoData.AcquisitionControl.ClearExposureComplete := THIS^.inoIoData.AcquisitionStatus.ExposureComplete;
		THIS^.inoIoData.AcquisitionControl.SetOffline := FALSE;
	
		THIS^.inoIoData.InspectionControl.EnableResultsBuffering := FALSE; 
		THIS^.inoIoData.InspectionControl.AcknowledgeInspectionResults := THIS^.inoIoData.InspectionStatus.ResultsValid;
		THIS^.inoIoData.InspectionControl.ExtendedUserDataSet := FALSE;
		THIS^.inoIoData.InspectionControl.ExecuteCommand := FALSE;
		THIS^.inoIoData.InspectionControl.ClearError := THIS^.inoIoData.InspectionStatus.Error;
		
		THIS^.inoIoData.CommandControl.Command:=0;

		_progress := _progress + 1;
	END_IF
	
	IF _progress = 2 THEN
		THIS^.Messenger.OnCondition(_infoTimer.Q).Warning('<#Waiting for the signal ExposureComplete to be reseted!#>').Pin(); 
		IF NOT THIS^.inoIoData.AcquisitionStatus.ExposureComplete THEN
			THIS^.inoIoData.AcquisitionControl.ClearExposureComplete := FALSE;
			CallTimers(FALSE);
			_progress := _progress + 1;
		END_IF
	END_IF
	
	IF _progress = 3 THEN
		THIS^.Messenger.OnCondition(_infoTimer.Q).Warning('<#Waiting for the signal ResultsValid to be reseted!#>').Pin(); 
		IF NOT THIS^.inoIoData.InspectionStatus.ResultsValid THEN
			THIS^.inoIoData.InspectionControl.AcknowledgeInspectionResults := FALSE;
			CallTimers(FALSE);
			_progress := _progress + 1;
		END_IF
	END_IF
	
	IF _progress = 4 THEN
		THIS^.Messenger.OnCondition(_infoTimer.Q).Warning('<#Waiting for the signal Error to be reseted!#>').Pin(); 
		IF NOT THIS^.inoIoData.InspectionStatus.Error THEN
			THIS^.inoIoData.InspectionControl.ClearError := FALSE;
			CallTimers(FALSE);
			_progress := _progress + 1;
		END_IF
	END_IF
	
	IF _progress = 5 THEN
		THIS^.Messenger.OnCondition(_infoTimer.Q).Warning('<#Waiting for the signal AcquisitionTriggerReady to be set!#>').Pin(); 
		_inspectionCompleted := THIS^.inoIoData.InspectionStatus.InspectionCompleted;
		IF THIS^.inoIoData.AcquisitionStatus.AcquisitionTriggerReady THEN
			CallTimers(FALSE);
			_progress := _progress + 1;
		END_IF
	END_IF
	
	IF _progress = 6 THEN
		THIS^.Messenger.OnCondition(_infoTimer.Q).Warning('<#Waiting for the signal AcquisitionTriggerAcknowledge to be set!#>').Pin(); 
		THIS^.inoIoData.AcquisitionControl.AcquisitionTrigger := TRUE;
		IF THIS^.inoIoData.AcquisitionStatus.AcquisitionTriggerAcknowledge THEN
			CallTimers(FALSE);
			_progress := _progress + 1;
		END_IF
	END_IF
	
	IF _progress = 7 THEN	
		THIS^.Messenger.OnCondition(_infoTimer.Q).Warning('<#Waiting for the signal InspectionCompleted to be toggled!#>').Pin(); 
		THIS^.inoIoData.AcquisitionControl.AcquisitionTrigger := FALSE;
		IF THIS^._inspectionCompleted <> THIS^.inoIoData.InspectionStatus.InspectionCompleted THEN
			CallTimers(FALSE);
			_progress := _progress + 1;
		END_IF
	END_IF

	IF _progress = 8 THEN
		THIS^.Messenger.OnCondition(_infoTimer.Q).Warning('<#Waiting for the signal ResultsValid to be set!#>').Pin(); 
		IF THIS^.inoIoData.InspectionStatus.ResultsValid THEN
			CallTimers(FALSE);
			_progress := _progress + 1;
		END_IF
	END_IF
	
	IF _progress = 9 THEN
		THIS^.Messenger.OnCondition(_infoTimer.Q).Warning('<#Waiting for the InspectionResults to be copied!#>').Pin(); 
		THIS^.inoResults.InspectionId := THIS^.inoIoData.ResultsData.InspectionID;
		THIS^.inoResults.ResultCode := THIS^.inoIoData.ResultsData.ResultCode;
		_size := THIS^.inoConfig.ResultDataSize;
		IF  Tc2_System.MEMCPY(srcAddr := ADR(THIS^.inoIoData.ResultsData.InspectionResults) , destAddr:= ADR(THIS^.inoResults.InspectionResults) ,  n:= _size) > 0 AND 
			Tc2_System.MEMSET(destAddr:= ADR(THIS^.inoResults.InspectionResults) + _size, fillByte:= 0 , n:= SIZEOF(THIS^.inoResults.InspectionResults) - _size)>0 THEN
			CallTimers(FALSE);
			_progress := _progress + 1;
		END_IF
	END_IF
	
	IF _progress = 10 THEN
		THIS^.inoIoData.AcquisitionControl.AcquisitionTrigger := FALSE;
		THIS^.inoIoData.InspectionControl.EnableResultsBuffering := FALSE;
		THIS^.inoIoData.InspectionControl.AcknowledgeInspectionResults := TRUE;
		THIS^.ThrowWhen(THIS^.inoIoData.InspectionStatus.Error);
		THIS^.DoneWhen(TRUE);
		_progress := 0;
	END_IF
	
	CallTimers(TRUE);
	
	THIS^.ThrowWhen(_errorTimer.Q OR _progress >4 AND THIS^.inoIoData.InspectionStatus.Error);	
END_IF

METHOD CallTimers
VAR_INPUT
	inValue : BOOL;
END_VAR
IF  __ISVALIDREF(inoConfig) AND THIS^.inoConfig.ErrorTime <> T#0S OR NOT inValue THEN  
_errorTimer(IN := inValue, PT := THIS^.inoConfig.ErrorTime);
END_IF;
IF  __ISVALIDREF(inoConfig) AND THIS^.inoConfig.InfoTime <>T#0S OR NOT inValue THEN  
_infoTimer(IN := inValue, PT := THIS^.inoConfig.InfoTime);
END_IF;
END_METHOD

{attribute 'hide'}
METHOD PUBLIC FB_init : BOOL
VAR_INPUT
	bInitRetains : BOOL; // if TRUE, the retain variables are initialized (warm start / cold start)
	bInCopyCode : BOOL;  // if TRUE, the instance afterwards gets moved into the copy code (online change)
	ParentObject : ITcoObject;
END_VAR
END_METHOD

(*~
	<docu>
		<summary>
			Executes when task is aborted.
		</summary>			
	</docu>	
~*)
METHOD PROTECTED OnAbort
THIS^.inoStatus.ActionDescription := '<#Trigger was aborted, while not yet completed!#>';
END_METHOD

(*~
	<docu>
		<summary>
			Executes when task reaches the ```Done``` state .
		</summary>			
	</docu>	
~*)
METHOD PROTECTED OnDone
THIS^.inoStatus.ActionDescription := '<#Trigger was completed successfully.#>';
END_METHOD

(*~
	<docu>
		<summary>
			Executes when task reaches the ```Error``` state.
			<para>
				Do not confuse with <see cref="PlcDocu.TcoCore.TcoTask.WhileError()"/>, that is called cyclically until '''Error''' state is left.
			</para>
		</summary>			
	</docu>	
~*)
METHOD PROTECTED OnError
THIS^.inoStatus.ActionDescription := '<#Trigger finished with error.#>';
END_METHOD

METHOD PROTECTED OnStart
THIS^.inoStatus.ActionDescription := '<#Trigger started.#>';
END_METHOD

(*~
	<docu>
		<summary>
			Restores this instance to the Ready state. Can be called explicitly or from within one of the restore mechanisms.
			<para>
				See also <see cref="PlcDocu.TcoCore.TcoTask.AutoRestorable()"/>
			</para>
		</summary>			
	</docu>	
~*)
METHOD Restore : ITcoRestorable
SUPER^.Restore();
_progress := 0;
CallTimers(FALSE);
Messenger.UnPin();
END_METHOD

END_FUNCTION_BLOCK

// ---- POUs/TcoInsight/v_5_x_x/Tasks/TcoInsightChangeJobByName_v_5_x_x.TcPOU
FUNCTION_BLOCK TcoInsightChangeJobByName_v_5_x_x EXTENDS TcoCore.TcoTask
VAR_IN_OUT
	inoIoData 	: TcoInsightIO_v_5_x_x;
    inoConfig 	: TcoInsightConfig_v_5_x_x;
	inoStatus 	: TcoInsightStatus_v_5_x_x;	
END_VAR
VAR
    {attribute addProperty Name "<#Job name#>"}
	_jobName : STRING;
END_VAR
VAR
    {attribute 'hide'} 
	_progress : INT := 0;
    {attribute 'hide'} 
	_infoTimer :  TON;
    {attribute 'hide'} 
	_errorTimer :  TON;
    {attribute 'hide'} 
	_varInfo : __SYSTEM.VAR_INFO;
    {attribute 'hide'} 
	_sb : TcoCore.StringBuilder;
END_VAR

IF Execute() THEN
	IF _progress = 0 THEN
		IF NOT __ISVALIDREF(inoIoData) THEN
			_varInfo :=__VARINFO(inoIoData);
			Messenger.Programming(_sb.Clear().Append('<#Invalid reference: #>').Append(_varInfo.Symbol).ToString()).Pin();
		ELSIF NOT __ISVALIDREF(inoConfig) THEN                                                  
			_varInfo :=__VARINFO(inoConfig);                                                    
			Messenger.Programming(_sb.Clear().Append('<#Invalid reference: #>').Append(_varInfo.Symbol).ToString()).Pin();
		ELSIF NOT __ISVALIDREF(inoStatus) THEN                                                  
			_varInfo :=__VARINFO(inoStatus);                                                    
			Messenger.Programming(_sb.Clear().Append('<#Invalid reference: #>').Append(_varInfo.Symbol).ToString()).Pin();
		ELSE
			_progress := _progress + 1;
		END_IF
	END_IF
	
	IF _progress = 1 THEN
		CallTimers(FALSE);
		IF _jobName='' THEN
			Messenger.Programming('<#Empty job name inserted!#>').Pin();
			THIS^.ThrowWhen(TRUE);
		ELSE	
			_progress := _progress + 1;
		END_IF
	END_IF
	
	IF _progress = 2 THEN
		THIS^.inoStatus.ActionDescription := _sb.Clear().Append('<#Change job by name (').Append(THIS^._jobName).Append(') is running.#>').ToString();  
		THIS^.Messenger.OnCondition(_infoTimer.Q).Warning('<#Waiting for the signal CommandExecuting to be reseted!#>').Pin(); 
		THIS^.inoIoData.InspectionControl.ExecuteCommand:=FALSE;
		THIS^.inoIoData.InspectionControl.ClearError:=FALSE;
		THIS^.inoIoData.AcquisitionControl.SetOffline := FALSE;
		IF NOT THIS^.inoIoData.InspectionStatus.CommandExecuting THEN
			CallTimers(FALSE);
			_progress := _progress + 1;
		END_IF
	END_IF
	
	IF _progress = 3 THEN	
		THIS^.Messenger.OnCondition(_infoTimer.Q).Warning('<#Waiting for the signal Online to be reseted!#>').Pin(); 
		THIS^.inoIoData.AcquisitionControl.SetOffline := TRUE;
		IF(NOT THIS^.inoIoData.AcquisitionStatus.Online) THEN
			CallTimers(FALSE);
			_progress := _progress + 1;
		END_IF
	END_IF

	IF _progress = 4 THEN	
		THIS^.Messenger.OnCondition(_infoTimer.Q).Warning('<#Waiting for the signal Error to be reseted!#>').Pin(); 
		THIS^.inoIoData.AcquisitionControl.SetOffline := TRUE;
		THIS^.inoIoData.InspectionControl.ExecuteCommand := FALSE;
		THIS^.inoIoData.InspectionControl.ClearError := THIS^.inoIoData.InspectionStatus.Error;
		IF NOT THIS^.inoIoData.InspectionStatus.Error THEN
			CallTimers(FALSE);
			_progress := _progress + 1;
		END_IF
	END_IF
	
	IF _progress = 5 THEN	
		THIS^.Messenger.OnCondition(_infoTimer.Q).Warning('<#Waiting for the Job name to be written to the User data!#>').Pin(); 
		THIS^.inoIoData.AcquisitionControl.SetOffline := TRUE;
		IF SetUserDataAsString(_jobName,0) THEN
			CallTimers(FALSE);
			_progress := _progress + 1;
		END_IF
	
	END_IF

	IF _progress = 6 THEN	
		THIS^.Messenger.OnCondition(_infoTimer.Q).Warning('<#Waiting for the signal ExtendedUserDataSetAcknowledge to be set!#>').Pin(); 
		THIS^.inoIoData.AcquisitionControl.SetOffline := TRUE;
		THIS^.inoIoData.InspectionControl.ExtendedUserDataSet := TRUE;
		IF(THIS^.inoIoData.InspectionStatus.ExtendedUserDataSetAcknowledge) THEN
			CallTimers(FALSE);
			_progress := _progress + 1;
		END_IF
	END_IF
		
	IF _progress = 7 THEN	
		THIS^.Messenger.OnCondition(_infoTimer.Q).Warning('<#Waiting for the signal ExtendedUserDataSetAcknowledge to be reseted!#>').Pin(); 
		THIS^.inoIoData.AcquisitionControl.SetOffline := TRUE;
		THIS^.inoIoData.InspectionControl.ExtendedUserDataSet := FALSE;
		IF(NOT THIS^.inoIoData.InspectionStatus.ExtendedUserDataSetAcknowledge) THEN
			CallTimers(FALSE);
			_progress := _progress + 1;
		END_IF
	END_IF

	IF _progress = 8 THEN	
		THIS^.Messenger.OnCondition(_infoTimer.Q).Warning('<#Waiting for the signal CommandComplete to be set!#>').Pin(); 
		THIS^.inoIoData.AcquisitionControl.SetOffline := TRUE;
		THIS^.inoIoData.CommandControl.Command := 16#4000;
		THIS^.inoIoData.InspectionControl.ExecuteCommand:=TRUE;
		
		IF(THIS^.inoIoData.InspectionStatus.CommandComplete AND NOT THIS^.inoIoData.InspectionStatus.CommandFailed) THEN
			CallTimers(FALSE);
			_progress := _progress + 1;
		ELSIF(THIS^.inoIoData.InspectionStatus.CommandComplete AND THIS^.inoIoData.InspectionStatus.CommandFailed AND NOT THIS^.inoIoData.InspectionStatus.CommandExecuting) THEN
			_progress := 20;
		END_IF;
	
	END_IF

	IF _progress = 9 THEN	
		THIS^.Messenger.OnCondition(_infoTimer.Q).Warning('<#Waiting for the signal CommandComplete to be reseted!#>').Pin(); 
		THIS^.inoIoData.AcquisitionControl.SetOffline := TRUE;
		THIS^.inoIoData.CommandControl.Command := 0;
		THIS^.inoIoData.InspectionControl.ExecuteCommand:=FALSE;
		IF(NOT THIS^.inoIoData.InspectionStatus.CommandComplete) THEN
			CallTimers(FALSE);
			_progress := _progress + 1;
		END_IF;
	END_IF

	IF _progress = 10 THEN	
		THIS^.Messenger.OnCondition(_infoTimer.Q).Warning('<#Waiting for the signal Online to be set!#>').Pin(); 
		THIS^.inoIoData.AcquisitionControl.SetOffline := FALSE;
		
		IF(THIS^.inoIoData.AcquisitionStatus.Online) THEN
			CallTimers(FALSE);
			_progress := _progress + 1;
		END_IF
	END_IF

	IF _progress = 11 THEN
		THIS^.inoStatus.CurrentJobName := _jobName;
		THIS^.inoIoData.InspectionControl.ExecuteCommand := FALSE;
		THIS^.inoIoData.AcquisitionControl.SetOffline := FALSE;
		THIS^.inoIoData.InspectionControl.ClearError := FALSE;
		THIS^.inoIoData.CommandControl.Command := 0;
		THIS^.ThrowWhen(FALSE);
		THIS^.DoneWhen(TRUE);
		_progress := 0;
	END_IF

	IF _progress = 20 THEN	
		Messenger.Error(CONCAT('<#Change job by name failed. Error code:#>',UINT_TO_STRING(inoIoData.InspectionStatus.ErrorCode))).Pin();
		THIS^.inoIoData.InspectionControl.ExecuteCommand := FALSE;
		THIS^.inoIoData.AcquisitionControl.SetOffline := FALSE;
		THIS^.inoIoData.CommandControl.Command := 0;
		THIS^.ThrowWhen(TRUE);
		THIS^.DoneWhen(FALSE);
	END_IF

	CallTimers(TRUE);
	
	THIS^.ThrowWhen(_errorTimer.Q);
	
END_IF

METHOD CallTimers
VAR_INPUT
	inValue : BOOL;
END_VAR
IF  __ISVALIDREF(inoConfig) AND THIS^.inoConfig.ErrorTime <> T#0S OR NOT inValue THEN  
_errorTimer(IN := inValue, PT := THIS^.inoConfig.ErrorTime);
END_IF;
IF  __ISVALIDREF(inoConfig) AND THIS^.inoConfig.InfoTime <>T#0S OR NOT inValue THEN  
_infoTimer(IN := inValue, PT := THIS^.inoConfig.InfoTime);
END_IF;
END_METHOD

{attribute 'hide'}
METHOD PUBLIC FB_init : BOOL
VAR_INPUT
	bInitRetains : BOOL; // if TRUE, the retain variables are initialized (warm start / cold start)
	bInCopyCode : BOOL;  // if TRUE, the instance afterwards gets moved into the copy code (online change)
	ParentObject : ITcoObject;
END_VAR
END_METHOD

METHOD INTERNAL InvokeWithParameters : ITcoTaskStatus
VAR_INPUT
    inJobName : STRING;
END_VAR
_jobName := inJobName;
InvokeWithParameters := THIS^.Invoke();
END_METHOD

(*~
	<docu>
		<summary>
			Executes when task is aborted.
		</summary>			
	</docu>	
~*)
METHOD PROTECTED OnAbort
THIS^.inoStatus.ActionDescription := _sb.Clear().Append('<#Change job by name (').Append(THIS^._jobName).Append(') aborted, while not yet finished.#>').ToString();
END_METHOD

(*~
	<docu>
		<summary>
			Executes when task reaches the ```Done``` state .
		</summary>			
	</docu>	
~*)
METHOD PROTECTED OnDone
THIS^.inoStatus.ActionDescription := _sb.Clear().Append('<#Change job by name (').Append(THIS^._jobName).Append(') was completed succesfully.#>').ToString();
END_METHOD

(*~
	<docu>
		<summary>
			Executes when task reaches the ```Error``` state.
			<para>
				Do not confuse with <see cref="PlcDocu.TcoCore.TcoTask.WhileError()"/>, that is called cyclically until '''Error''' state is left.
			</para>
		</summary>			
	</docu>	
~*)
METHOD PROTECTED OnError
THIS^.inoStatus.ActionDescription := _sb.Clear().Append('<#Change job by name (').Append(THIS^._jobName).Append(') finished with error.#>').ToString();
END_METHOD

METHOD PROTECTED OnStart
THIS^.inoStatus.ActionDescription := _sb.Clear().Append('<#Change job by name (').Append(THIS^._jobName).Append(') started.#>').ToString();
END_METHOD

(*~
	<docu>
		<summary>
			Restores this instance to the Ready state. Can be called explicitly or from within one of the restore mechanisms.
			<para>
				See also <see cref="PlcDocu.TcoCore.TcoTask.AutoRestorable()"/>
			</para>
		</summary>			
	</docu>	
~*)
METHOD Restore : ITcoRestorable
SUPER^.Restore();
_progress := 0;
CallTimers(FALSE);
Messenger.UnPin();
END_METHOD

METHOD INTERNAL SetUserDataAsString : BOOL
VAR_INPUT
	inValue : STRING;
	inPosition : UINT;	
END_VAR
VAR
	_index : UINT;
	_size : UINT;
	_bufferSize : UINT; 
END_VAR
SetUserDataAsString := FALSE;

_size := LEN(inValue);

//_bufferSize := SIZEOF(inoUserData.UserData)/SIZEOF(inoUserData.UserData[0]);
_bufferSize := SIZEOF(THIS^.inoIoData.UserData.UserData)/SIZEOF(THIS^.inoIoData.UserData.UserData[0]);

IF (inPosition +_size) > THIS^.inoConfig.UserDataSize THEN
	Messenger.Programming('<#Index of UserData in method SetUserDataAsString exceeds the size hardware structure mapped!#>');
	RETURN;
END_IF

IF (inPosition +_size) > _bufferSize THEN
	Messenger.Programming('<#Index of UserData in method SetUserDataAsString exceeds the defined size!#>');
	RETURN;
END_IF

FOR	_index := 1 TO _size BY 1 DO	
	THIS^.inoIoData.UserData.UserData[inPosition + _index-1] := F_ToASC(MID(inValue,1,_index));
END_FOR;

FOR	_index := inPosition +_size TO _bufferSize BY 1 DO	
	THIS^.inoIoData.UserData.UserData[_index] := 0;
END_FOR;

SetUserDataAsString := TRUE;
END_METHOD

END_FUNCTION_BLOCK

// ---- POUs/TcoInsight/v_5_x_x/Tasks/TcoInsightChangeJobByNumber_v_5_x_x.TcPOU
FUNCTION_BLOCK TcoInsightChangeJobByNumber_v_5_x_x EXTENDS TcoCore.TcoTask
VAR_IN_OUT
	inoIoData 	: TcoInsightIO_v_5_x_x;
    inoConfig 	: TcoInsightConfig_v_5_x_x;
	inoStatus 	: TcoInsightStatus_v_5_x_x;	
END_VAR
VAR
   {attribute addProperty Name "<#Job number#>"}
	_jobNumber : UINT;
END_VAR
VAR
    {attribute 'hide'} 
	_progress : INT := 0;
    {attribute 'hide'} 
	_infoTimer :  TON;
    {attribute 'hide'} 
	_errorTimer :  TON;
    {attribute 'hide'} 
	_varInfo : __SYSTEM.VAR_INFO;
    {attribute 'hide'} 
	_sb : TcoCore.StringBuilder;
END_VAR

IF Execute() THEN
	IF _progress = 0 THEN
		IF NOT __ISVALIDREF(inoIoData) THEN
			_varInfo :=__VARINFO(inoIoData);
			Messenger.Programming(_sb.Clear().Append('<#Invalid reference: #>').Append(_varInfo.Symbol).ToString()).Pin();
		ELSIF NOT __ISVALIDREF(inoConfig) THEN                                                  
			_varInfo :=__VARINFO(inoConfig);                                                    
			Messenger.Programming(_sb.Clear().Append('<#Invalid reference: #>').Append(_varInfo.Symbol).ToString()).Pin();
		ELSIF NOT __ISVALIDREF(inoStatus) THEN                                                  
			_varInfo :=__VARINFO(inoStatus);                                                    
			Messenger.Programming(_sb.Clear().Append('<#Invalid reference: #>').Append(_varInfo.Symbol).ToString()).Pin();
		ELSE
			_progress := _progress + 1;
		END_IF
	END_IF
	
	IF _progress = 1 THEN
		CallTimers(FALSE);
		IF _jobNumber > inoConfig.MaxJobNumber THEN
			Messenger.Programming(_sb.Clear().Append('<#Job number (').Append(UINT_TO_STRING(_jobNumber)).Append(') is greater than the maximal value of ').Append(UINT_TO_STRING(inoConfig.MaxJobNumber)).Append('!#>').ToString()).Pin();
			THIS^.ThrowWhen(TRUE);
		ELSE	
			_progress := _progress + 1;
		END_IF
	END_IF
	
	IF _progress = 2 THEN
		THIS^.inoStatus.ActionDescription := _sb.Clear().Append('<#Change job by number (').Append(UINT_TO_STRING(THIS^._jobNumber)).Append(') is running.#>').ToString(); 
		THIS^.Messenger.OnCondition(_infoTimer.Q).Warning('<#Waiting for the signal CommandExecuting to be reseted!#>').Pin(); 
		THIS^.inoIoData.InspectionControl.ExecuteCommand:=FALSE;
		THIS^.inoIoData.InspectionControl.ClearError:=FALSE;
		THIS^.inoIoData.AcquisitionControl.SetOffline := FALSE;
		IF NOT THIS^.inoIoData.InspectionStatus.CommandExecuting THEN
			CallTimers(FALSE);
			_progress := _progress + 1;
		END_IF
	END_IF
	
	IF _progress = 3 THEN	
		THIS^.Messenger.OnCondition(_infoTimer.Q).Warning('<#Waiting for the signal Online to be reseted!#>').Pin(); 
		THIS^.inoIoData.AcquisitionControl.SetOffline := TRUE;
		IF(NOT THIS^.inoIoData.AcquisitionStatus.Online) THEN
			CallTimers(FALSE);
			_progress := _progress + 1;
		END_IF
	END_IF

	IF _progress = 4 THEN	
		THIS^.Messenger.OnCondition(_infoTimer.Q).Warning('<#Waiting for the signal Error to be reseted!#>').Pin(); 
		THIS^.inoIoData.AcquisitionControl.SetOffline := TRUE;
		THIS^.inoIoData.InspectionControl.ExecuteCommand := FALSE;
		THIS^.inoIoData.InspectionControl.ClearError := THIS^.inoIoData.InspectionStatus.Error;
		IF NOT THIS^.inoIoData.InspectionStatus.Error THEN
			CallTimers(FALSE);
			_progress := _progress + 1;
		END_IF
	END_IF
	
	IF _progress = 5 THEN	
		THIS^.Messenger.OnCondition(_infoTimer.Q).Warning('<#Waiting for the signal CommandComplete to be set!#>').Pin(); 
		THIS^.inoIoData.AcquisitionControl.SetOffline := TRUE;
		THIS^.inoIoData.CommandControl.Command := _jobNumber;
		THIS^.inoIoData.InspectionControl.ExecuteCommand:=TRUE;
		
		IF(THIS^.inoIoData.InspectionStatus.CommandComplete AND NOT THIS^.inoIoData.InspectionStatus.CommandFailed) THEN
			CallTimers(FALSE);
			_progress := _progress + 1;
		ELSIF(THIS^.inoIoData.InspectionStatus.CommandComplete AND THIS^.inoIoData.InspectionStatus.CommandFailed AND NOT THIS^.inoIoData.InspectionStatus.CommandExecuting) THEN
			_progress := 20;
		END_IF;
	
	END_IF

	IF _progress = 6 THEN	
		THIS^.Messenger.OnCondition(_infoTimer.Q).Warning('<#Waiting for the signal CommandComplete to be reseted!#>').Pin(); 
		THIS^.inoIoData.AcquisitionControl.SetOffline := TRUE;
		THIS^.inoIoData.CommandControl.Command := 0;
		THIS^.inoIoData.InspectionControl.ExecuteCommand:=FALSE;
		IF(NOT THIS^.inoIoData.InspectionStatus.CommandComplete) THEN
			CallTimers(FALSE);
			_progress := _progress + 1;
		END_IF;
	END_IF

	IF _progress = 7 THEN	
		THIS^.Messenger.OnCondition(_infoTimer.Q).Warning('<#Waiting for the signal Online to be set!#>').Pin(); 
		THIS^.inoIoData.AcquisitionControl.SetOffline := FALSE;
		
		IF(THIS^.inoIoData.AcquisitionStatus.Online) THEN
			CallTimers(FALSE);
			_progress := _progress + 1;
		END_IF
	END_IF

	IF _progress = 8 THEN
		THIS^.inoStatus.CurrentJobNumber := UINT_TO_INT(_jobNumber);
		THIS^.inoIoData.InspectionControl.ExecuteCommand := FALSE;
		THIS^.inoIoData.AcquisitionControl.SetOffline := FALSE;
		THIS^.inoIoData.InspectionControl.ClearError := FALSE;
		THIS^.inoIoData.CommandControl.Command := 0;
		THIS^.ThrowWhen(FALSE);
		THIS^.DoneWhen(TRUE);
		_progress := 0;
	END_IF

	IF _progress = 20 THEN	
		Messenger.Error(_sb.Clear().Append('<#Change job by number failed. Error code:#>').Append(UINT_TO_STRING(inoIoData.InspectionStatus.ErrorCode)).ToString()).Pin();
		THIS^.inoIoData.InspectionControl.ExecuteCommand := FALSE;
		THIS^.inoIoData.AcquisitionControl.SetOffline := FALSE;
		THIS^.inoIoData.CommandControl.Command := 0;
		THIS^.ThrowWhen(TRUE);
		THIS^.DoneWhen(FALSE);
	END_IF

	CallTimers(TRUE);
	
	THIS^.ThrowWhen(_errorTimer.Q);
	
END_IF

METHOD CallTimers
VAR_INPUT
	inValue : BOOL;
END_VAR
IF  __ISVALIDREF(inoConfig) AND THIS^.inoConfig.ErrorTime <> T#0S OR NOT inValue THEN  
_errorTimer(IN := inValue, PT := THIS^.inoConfig.ErrorTime);
END_IF;
IF  __ISVALIDREF(inoConfig) AND THIS^.inoConfig.InfoTime <>T#0S OR NOT inValue THEN  
_infoTimer(IN := inValue, PT := THIS^.inoConfig.InfoTime);
END_IF;
END_METHOD

{attribute 'hide'}
METHOD PUBLIC FB_init : BOOL
VAR_INPUT
	bInitRetains : BOOL; // if TRUE, the retain variables are initialized (warm start / cold start)
	bInCopyCode : BOOL;  // if TRUE, the instance afterwards gets moved into the copy code (online change)
	ParentObject : ITcoObject;
END_VAR
END_METHOD

METHOD INTERNAL InvokeWithParameters : ITcoTaskStatus
VAR_INPUT
	inJobNumber : UINT;
END_VAR
_jobNumber := inJobNumber;
InvokeWithParameters := THIS^.Invoke();
END_METHOD

(*~
	<docu>
		<summary>
			Executes when task is aborted.
		</summary>			
	</docu>	
~*)
METHOD PROTECTED OnAbort
THIS^.inoStatus.ActionDescription := _sb.Clear().Append('<#Change job by number (').Append(UINT_TO_STRING(THIS^._jobNumber)).Append(') aborted, while not yet finished.#>').ToString();
END_METHOD

(*~
	<docu>
		<summary>
			Executes when task reaches the ```Done``` state .
		</summary>			
	</docu>	
~*)
METHOD PROTECTED OnDone
THIS^.inoStatus.ActionDescription := _sb.Clear().Append('<#Change job by number (').Append(UINT_TO_STRING(THIS^._jobNumber)).Append(') was completed succesfully.#>').ToString();
END_METHOD

(*~
	<docu>
		<summary>
			Executes when task reaches the ```Error``` state.
			<para>
				Do not confuse with <see cref="PlcDocu.TcoCore.TcoTask.WhileError()"/>, that is called cyclically until '''Error''' state is left.
			</para>
		</summary>			
	</docu>	
~*)
METHOD PROTECTED OnError
THIS^.inoStatus.ActionDescription := _sb.Clear().Append('<#Change job by number (').Append(UINT_TO_STRING(THIS^._jobNumber)).Append(') finished with error.#>').ToString();
END_METHOD

METHOD PROTECTED OnStart
THIS^.inoStatus.ActionDescription := _sb.Clear().Append('<#Change job by number (').Append(UINT_TO_STRING(THIS^._jobNumber)).Append(') started.#>').ToString();
END_METHOD

(*~
	<docu>
		<summary>
			Restores this instance to the Ready state. Can be called explicitly or from within one of the restore mechanisms.
			<para>
				See also <see cref="PlcDocu.TcoCore.TcoTask.AutoRestorable()"/>
			</para>
		</summary>			
	</docu>	
~*)
METHOD Restore : ITcoRestorable
SUPER^.Restore();
_progress := 0;
CallTimers(FALSE);
Messenger.UnPin();
END_METHOD

END_FUNCTION_BLOCK

// ---- POUs/TcoInsight/v_5_x_x/Tasks/TcoInsightClearInspectionResults_v_5_x_x.TcPOU
FUNCTION_BLOCK TcoInsightClearInspectionResults_v_5_x_x EXTENDS TcoCore.TcoTask
VAR_IN_OUT
	inoIoData	: TcoInsightIO_v_5_x_x;
    inoConfig	: TcoInsightConfig_v_5_x_x;
	inoStatus	: TcoInsightStatus_v_5_x_x;	
	inoResults 	: TcoInsightResults_v_5_x_x;
END_VAR
VAR
    {attribute 'hide'} 
	_progress : INT := 0;
    {attribute 'hide'} 
	_infoTimer :  TON;
    {attribute 'hide'} 
	_errorTimer :  TON;
    {attribute 'hide'} 
	_varInfo : __SYSTEM.VAR_INFO;
    {attribute 'hide'} 
	_sb : TcoCore.StringBuilder;
END_VAR

IF Execute() THEN
	IF _progress = 0 THEN
		IF NOT __ISVALIDREF(inoIoData) THEN
			_varInfo :=__VARINFO(inoIoData);
			Messenger.Programming(_sb.Clear().Append('<#Invalid reference: #>').Append(_varInfo.Symbol).ToString()).Pin();
		ELSIF NOT __ISVALIDREF(inoConfig) THEN                                                  
			_varInfo :=__VARINFO(inoConfig);                                                    
			Messenger.Programming(_sb.Clear().Append('<#Invalid reference: #>').Append(_varInfo.Symbol).ToString()).Pin();
		ELSIF NOT __ISVALIDREF(inoStatus) THEN                                                  
			_varInfo :=__VARINFO(inoStatus);                                                    
			Messenger.Programming(_sb.Clear().Append('<#Invalid reference: #>').Append(_varInfo.Symbol).ToString()).Pin();
		ELSIF NOT __ISVALIDREF(inoResults) THEN                                              
			_varInfo :=__VARINFO(inoResults);                                                
			Messenger.Programming(_sb.Clear().Append('<#Invalid reference: #>').Append(_varInfo.Symbol).ToString()).Pin();
		ELSE
			_progress := _progress + 1;
		END_IF
	END_IF
	
	IF _progress = 1 THEN
		THIS^.inoStatus.ActionDescription := '<#Clearing result data running.#>'; 
		CallTimers(FALSE);
		_progress := _progress + 1;
	END_IF
	
	IF _progress = 2 THEN
		THIS^.inoIoData.AcquisitionControl.AcquisitionTriggerEnable := FALSE;
		THIS^.inoIoData.AcquisitionControl.AcquisitionTrigger := FALSE;
		THIS^.inoIoData.InspectionControl.AcknowledgeInspectionResults := TRUE;
		THIS^.Messenger.OnCondition(_infoTimer.Q).Warning('<#Waiting for the result data cleared!#>').Pin();
		THIS^.inoResults.InspectionId := 0;
		THIS^.inoResults.ResultCode := 0;
		IF Tc2_System.MEMSET(destAddr:= ADR(THIS^.inoResults.InspectionResults) , fillByte:= 0 , n:= SIZEOF(THIS^.inoResults.InspectionResults)) >0 THEN
			CallTimers(FALSE);
			_progress := _progress + 1;
		END_IF
	END_IF
	
	IF _progress = 3 THEN
		THIS^.Messenger.OnCondition(_infoTimer.Q).Warning('<#Waiting for the signal ResultsValid reseted!#>').Pin(); 
		IF NOT THIS^.inoIoData.InspectionStatus.ResultsValid THEN
			CallTimers(FALSE);
			_progress := _progress + 1;
		END_IF
	END_IF
	
	IF _progress = 4 THEN
		THIS^.inoIoData.InspectionControl.AcknowledgeInspectionResults := FALSE;
		THIS^.DoneWhen(TRUE);
		CallTimers(FALSE);
		_progress := 0;
	END_IF
	
	CallTimers(TRUE);
	
	THIS^.ThrowWhen(_errorTimer.Q);
END_IF

METHOD CallTimers
VAR_INPUT
	inValue : BOOL;
END_VAR
IF  __ISVALIDREF(inoConfig) AND THIS^.inoConfig.ErrorTime <> T#0S OR NOT inValue THEN  
_errorTimer(IN := inValue, PT := THIS^.inoConfig.ErrorTime);
END_IF;
IF  __ISVALIDREF(inoConfig) AND THIS^.inoConfig.InfoTime <>T#0S OR NOT inValue THEN  
_infoTimer(IN := inValue, PT := THIS^.inoConfig.InfoTime);
END_IF;
END_METHOD

{attribute 'hide'}
METHOD PUBLIC FB_init : BOOL
VAR_INPUT
	bInitRetains : BOOL; // if TRUE, the retain variables are initialized (warm start / cold start)
	bInCopyCode : BOOL;  // if TRUE, the instance afterwards gets moved into the copy code (online change)
	ParentObject : ITcoObject;
END_VAR
END_METHOD

(*~
	<docu>
		<summary>
			Executes when task is aborted.
		</summary>			
	</docu>	
~*)
METHOD PROTECTED OnAbort
THIS^.inoStatus.ActionDescription := '<#Clearing of the inspection results aborted, while not yet finished.#>';
END_METHOD

(*~
	<docu>
		<summary>
			Executes when task reaches the ```Done``` state .
		</summary>			
	</docu>	
~*)
METHOD PROTECTED OnDone
THIS^.inoStatus.ActionDescription := '<#Clearing of the inspection results was completed succesfully.#>';
END_METHOD

(*~
	<docu>
		<summary>
			Executes when task reaches the ```Error``` state.
			<para>
				Do not confuse with <see cref="PlcDocu.TcoCore.TcoTask.WhileError()"/>, that is called cyclically until '''Error''' state is left.
			</para>
		</summary>			
	</docu>	
~*)
METHOD PROTECTED OnError
THIS^.inoStatus.ActionDescription := '<#Clearing of the inspection results finished with error.#>';
END_METHOD

METHOD PROTECTED OnStart
THIS^.inoStatus.ActionDescription := '<#Clearing of the inspection results started.#>';
END_METHOD

(*~
	<docu>
		<summary>
			Restores this instance to the Ready state. Can be called explicitly or from within one of the restore mechanisms.
			<para>
				See also <see cref="PlcDocu.TcoCore.TcoTask.AutoRestorable()"/>
			</para>
		</summary>			
	</docu>	
~*)
METHOD Restore : ITcoRestorable
SUPER^.Restore();
_progress := 0;
CallTimers(FALSE);
Messenger.UnPin();
END_METHOD

END_FUNCTION_BLOCK

// ---- POUs/TcoInsight/v_5_x_x/Tasks/TcoInsightSoftEvent_v_5_x_x.TcPOU
FUNCTION_BLOCK TcoInsightSoftEvent_v_5_x_x EXTENDS TcoCore.TcoTask
VAR_IN_OUT
	inoIoData	: TcoInsightIO_v_5_x_x;
    inoConfig	: TcoInsightConfig_v_5_x_x;
	inoStatus	: TcoInsightStatus_v_5_x_x;	
END_VAR
VAR
   {attribute addProperty Name "<#Soft event number#>"}
	_softEventNumber : UINT;
END_VAR
VAR
    {attribute 'hide'} 
	_progress : INT := 0;
    {attribute 'hide'} 
	_infoTimer :  TON;
    {attribute 'hide'} 
	_errorTimer :  TON;
    {attribute 'hide'} 
	_varInfo : __SYSTEM.VAR_INFO;
    {attribute 'hide'} 
	_sb : TcoCore.StringBuilder;
    {attribute 'hide'} 
	_inspectionCompleted : BOOL;
END_VAR

IF Execute() THEN
	IF _progress = 0 THEN
		IF NOT __ISVALIDREF(inoIoData) THEN
			_varInfo :=__VARINFO(inoIoData);
			Messenger.Programming(_sb.Clear().Append('<#Invalid reference: #>').Append(_varInfo.Symbol).ToString()).Pin();
		ELSIF NOT __ISVALIDREF(inoConfig) THEN                                                  
			_varInfo :=__VARINFO(inoConfig);                                                    
			Messenger.Programming(_sb.Clear().Append('<#Invalid reference: #>').Append(_varInfo.Symbol).ToString()).Pin();
		ELSIF NOT __ISVALIDREF(inoStatus) THEN                                                  
			_varInfo :=__VARINFO(inoStatus);                                                    
			Messenger.Programming(_sb.Clear().Append('<#Invalid reference: #>').Append(_varInfo.Symbol).ToString()).Pin();
		ELSE
			_progress := _progress + 1;
		END_IF
	END_IF
	
	IF _progress = 1 THEN
		CallTimers(FALSE);
		IF _softEventNumber > 7 THEN
			Messenger.Programming(_sb.Clear().Append('<#SoftEvent number: (').Append(UINT_TO_STRING(_softEventNumber)).Append(') is greater than the maximal value of 7!#>').ToString()).Pin();
			THIS^.ThrowWhen(TRUE);
		ELSE	
			_progress := _progress + 1;
		END_IF
	END_IF
	
	IF _progress = 2 THEN
		THIS^.inoStatus.ActionDescription := _sb.Clear().Append('<#SoftEvent (number: ').Append(UINT_TO_STRING(THIS^._softEventNumber)).Append(') is running.#>').ToString();
		CallTimers(FALSE);
		_progress := _progress + 1;
	END_IF
	
	IF _progress = 3 THEN
		THIS^.Messenger.OnCondition(_infoTimer.Q).Warning(_sb.Clear().Append('<#Waiting for the signal TriggerSoftEvent[').Append(UINT_TO_STRING(THIS^._softEventNumber)).Append('] to be set!#>').ToString()).Pin(); 
		THIS^.inoIoData.SoftEventControl.TriggerSoftEvent[_softEventNumber] := TRUE;
		IF THIS^.inoIoData.SoftEventControl.TriggerSoftEventAcknowledge[_softEventNumber] THEN
			CallTimers(FALSE);
			_progress := _progress + 1;
		END_IF
	END_IF
	
	IF _progress = 4 THEN
		THIS^.Messenger.OnCondition(_infoTimer.Q).Warning(_sb.Clear().Append('<#Waiting for the signal TriggerSoftEvent[').Append(UINT_TO_STRING(THIS^._softEventNumber)).Append('] to be reseted!#>').ToString()).Pin(); 
		THIS^.inoIoData.SoftEventControl.TriggerSoftEvent[_softEventNumber] := FALSE;
		IF NOT THIS^.inoIoData.SoftEventControl.TriggerSoftEventAcknowledge[_softEventNumber] THEN
			CallTimers(FALSE);
			_progress := _progress + 1;
		END_IF
	END_IF

	IF _progress = 5 THEN
		THIS^.DoneWhen(TRUE);
		_progress := 0;
	END_IF
	
	CallTimers(TRUE);
	
	THIS^.ThrowWhen(_errorTimer.Q);
	
END_IF

METHOD CallTimers
VAR_INPUT
	inValue : BOOL;
END_VAR
IF  __ISVALIDREF(inoConfig) AND THIS^.inoConfig.ErrorTime <> T#0S OR NOT inValue THEN  
_errorTimer(IN := inValue, PT := THIS^.inoConfig.ErrorTime);
END_IF;
IF  __ISVALIDREF(inoConfig) AND THIS^.inoConfig.InfoTime <>T#0S OR NOT inValue THEN  
_infoTimer(IN := inValue, PT := THIS^.inoConfig.InfoTime);
END_IF;
END_METHOD

{attribute 'hide'}
METHOD PUBLIC FB_init : BOOL
VAR_INPUT
	bInitRetains : BOOL; // if TRUE, the retain variables are initialized (warm start / cold start)
	bInCopyCode : BOOL;  // if TRUE, the instance afterwards gets moved into the copy code (online change)
	ParentObject : ITcoObject;
END_VAR
END_METHOD

METHOD INTERNAL InvokeWithParameters : ITcoTaskStatus
VAR_INPUT
    inSoftEventNumber : UINT;
END_VAR
_softEventNumber := inSoftEventNumber;
InvokeWithParameters := THIS^.Invoke();
END_METHOD

(*~
	<docu>
		<summary>
			Executes when task is aborted.
		</summary>			
	</docu>	
~*)
METHOD PROTECTED OnAbort
THIS^.inoStatus.ActionDescription := _sb.Clear().Append('<#SoftEvent (number: ').Append(UINT_TO_STRING(THIS^._softEventNumber)).Append(') was aborted, while not yet completed.#>').ToString();
END_METHOD

(*~
	<docu>
		<summary>
			Executes when task reaches the ```Done``` state .
		</summary>			
	</docu>	
~*)
METHOD PROTECTED OnDone
THIS^.inoStatus.ActionDescription := _sb.Clear().Append('<#SoftEvent (number: ').Append(UINT_TO_STRING(THIS^._softEventNumber)).Append(') was completed successfully.#>').ToString();
END_METHOD

(*~
	<docu>
		<summary>
			Executes when task reaches the ```Error``` state.
			<para>
				Do not confuse with <see cref="PlcDocu.TcoCore.TcoTask.WhileError()"/>, that is called cyclically until '''Error''' state is left.
			</para>
		</summary>			
	</docu>	
~*)
METHOD PROTECTED OnError
THIS^.inoStatus.ActionDescription := _sb.Clear().Append('<#SoftEvent (number: ').Append(UINT_TO_STRING(THIS^._softEventNumber)).Append(') finished with error.#>').ToString();
END_METHOD

METHOD PROTECTED OnStart
THIS^.inoStatus.ActionDescription := _sb.Clear().Append('<#SoftEvent (number: ').Append(UINT_TO_STRING(THIS^._softEventNumber)).Append(') started.#>').ToString();
END_METHOD

(*~
	<docu>
		<summary>
			Restores this instance to the Ready state. Can be called explicitly or from within one of the restore mechanisms.
			<para>
				See also <see cref="PlcDocu.TcoCore.TcoTask.AutoRestorable()"/>
			</para>
		</summary>			
	</docu>	
~*)
METHOD Restore : ITcoRestorable
SUPER^.Restore();
_progress := 0;
CallTimers(FALSE);
Messenger.UnPin();
END_METHOD

END_FUNCTION_BLOCK

// ---- POUs/TcoInsight/v_5_x_x/TcoInsight_v_5_x_x.TcPOU
FUNCTION_BLOCK TcoInsight_v_5_x_x  EXTENDS TcoIo.TcoPnIoComponent 
VAR_IN_OUT
	inoIoData : TcoInsightIO_v_5_x_x;
END_VAR

VAR
	{attribute addProperty Name "<#Config#>"}
    _config : TcoInsightConfig_v_5_x_x;
	{attribute addProperty Name "<#Status#>"}
	_status : TcoInsightStatus_v_5_x_x;	
END_VAR

VAR
	{attribute addProperty Name "<#UserData#>"}
	_userData 	: TcoInsightUser_v_5_x_x;
	{attribute addProperty Name "<#Results#>"}
	_results : TcoInsightResults_v_5_x_x;
END_VAR

VAR
	{attribute 'hide'}
    _taskEnabled : BOOL;
	{attribute addProperty Name "<#Restore#>"}
    _restoreTask : TcoCore.TcoTask(THIS^);
	{attribute addProperty Name "<#Update signal states#>"}
    _updateSignalStatesTask : TcoCore.TcoTask(THIS^);
	{attribute addProperty Name "<#Change job by number#>"}
    _changeJobByNumberTask : TcoInsightChangeJobByNumber_v_5_x_x(THIS^);
	{attribute addProperty Name "<#Change job by name#>"}
    _changeJobByNameTask : TcoInsightChangeJobByName_v_5_x_x(THIS^);
	{attribute addProperty Name "<#Clear inspection results#>"}
    _clearInspectionResultsTask : TcoInsightClearInspectionResults_v_5_x_x(THIS^);
	{attribute addProperty Name "<#Set user data#>"}
    _setUserDataTask : TcoInsightSetUserData_v_5_x_x(THIS^);
	{attribute addProperty Name "<#Clear user data#>"}
    _clearUserDataTask : TcoInsightClearUserData_v_5_x_x(THIS^);
	{attribute addProperty Name "<#Soft event#>"}
    _softEventTask : TcoInsightSoftEvent_v_5_x_x(THIS^);
	{attribute addProperty Name "<#Trigger#>"}
    _triggerTask : TcoInsightTrigger_v_5_x_x(THIS^);
END_VAR
VAR
    {attribute 'hide'} 
	_varInfo : __SYSTEM.VAR_INFO;
    {attribute 'hide'} 
	_sb : TcoCore.StringBuilder;
END_VAR

IF InvalidReference() THEN
    RETURN;
END_IF

SUPER^(inPnIoBoxState := THIS^.inoIoData.PnIoBoxState,inPnIoBoxDiag := THIS^.inoIoData.PnIoBoxDiag);

IF NOT SUPER^.ProfinetReady THEN
	THIS^._status.ActionDescription := '<#Not ready for operation by means of Profinet network!#>';	
END_IF

IF SUPER^.ProfinetReady AND THIS^._status.ActionDescription = '<#Not ready for operation by means of Profinet network!#>' THEN
	THIS^._status.ActionDescription := '<#Ready for operation!#>';	
END_IF

CheckIfOnline();

//*************RESTORE********************
_taskEnabled := TRUE;
_restoreTask.Enabled := _taskEnabled;
IF _restoreTask.Execute() THEN
	Restore();
//	UpdateSignalStates();
END_IF
//****************************************

//*************UPDATE*********************
IF _config.UpdateStatesPermanently THEN
	UpdateSignalStates();
END_IF;

_taskEnabled:=SUPER^.ProfinetReady;
_taskEnabled := _taskEnabled AND NOT _restoreTask.Busy ;
_updateSignalStatesTask.Enabled := _taskEnabled;
IF _updateSignalStatesTask.Execute() THEN
	UpdateSignalStates();
END_IF
//****************************************

//*************CHANGE*JOB*BY*NUMBER*******
_taskEnabled:=SUPER^.ProfinetReady;
_taskEnabled := _taskEnabled AND NOT _updateSignalStatesTask.Busy;
_changeJobByNumberTask.Enabled := _taskEnabled;
_changeJobByNumberTask(inoIoData := THIS^.inoIoData,inoConfig := THIS^._config,inoStatus := THIS^._status);
//****************************************

//*************CHANGE*JOB*BY*NAME*********
_taskEnabled:=SUPER^.ProfinetReady;
_taskEnabled := _taskEnabled AND NOT _changeJobByNumberTask.Busy;
_changeJobByNameTask.Enabled := _taskEnabled;
_changeJobByNameTask(inoIoData := THIS^.inoIoData,inoConfig := THIS^._config,inoStatus := THIS^._status);
//****************************************

//*************CLEAR*DATA*****************
_taskEnabled:=SUPER^.ProfinetReady;
_taskEnabled := _taskEnabled AND NOT _changeJobByNameTask.Busy;
_clearInspectionResultsTask.Enabled := _taskEnabled;
_clearInspectionResultsTask(inoIoData := THIS^.inoIoData,inoConfig := THIS^._config,inoStatus := THIS^._status,inoResults := THIS^._results);
//****************************************

//*************CLEAR USER DATA*****************
_taskEnabled:=SUPER^.ProfinetReady;
_taskEnabled := _taskEnabled AND NOT _setUserDataTask.Busy  ;
_clearUserDataTask.Enabled := _taskEnabled;
_clearUserDataTask(inoIoData := THIS^.inoIoData,inoConfig := THIS^._config,inoStatus := THIS^._status,inoUserData := THIS^._userData);
//****************************************

//*************SET USER DATA*****************
_taskEnabled:=SUPER^.ProfinetReady;
_taskEnabled := _taskEnabled AND NOT _changeJobByNameTask.Busy AND NOT _clearInspectionResultsTask.Busy AND NOT _triggerTask.Busy ;
_setUserDataTask.Enabled := _taskEnabled;
_setUserDataTask(inoIoData := THIS^.inoIoData,inoConfig := THIS^._config,inoStatus := THIS^._status,inoUserData := THIS^._userData);
//****************************************

//*************SOFT*EVENT*****************
_taskEnabled:=SUPER^.ProfinetReady;
_taskEnabled := _taskEnabled AND THIS^.inoIoData.AcquisitionStatus.Online AND NOT _clearInspectionResultsTask.Busy AND NOT _setUserDataTask.Busy;
_softEventTask.Enabled := _taskEnabled;
_softEventTask(inoIoData := THIS^.inoIoData,inoConfig := THIS^._config,inoStatus := THIS^._status);
//****************************************

//*************TRIGGER********************
_taskEnabled:=SUPER^.ProfinetReady;
_taskEnabled := _taskEnabled AND NOT _clearInspectionResultsTask.Busy AND NOT _setUserDataTask.Busy;
_triggerTask.Enabled :=  _taskEnabled;
_triggerTask(inoIoData := THIS^.inoIoData,inoConfig := THIS^._config,inoStatus := THIS^._status,inoResults := THIS^._results);
//****************************************

(*~
	<docu>
		<summary>
			Clears the inspection results. 		
		</summary>			
	</docu>	
~*)
METHOD ClearInspectionResults : TcoCore.ITcoTaskStatus
ClearInspectionResults := THIS^._clearInspectionResultsTask.Invoke();
END_METHOD

(*~
	<docu>
		<summary>
			Gets the `ClearResultDataTask` task that controls clearing of the results data. 		
		</summary>			
	</docu>	
~*)
PROPERTY ClearInspectionResultsTask : TcoCore.ITcoTaskStatus
GET
ClearInspectionResultsTask := THIS^._clearInspectionResultsTask;
END_GET
END_PROPERTY

(*~
	<docu>
		<summary>
			Clears user data. 		
		</summary>			
	</docu>	
~*)
METHOD ClearUserData : TcoCore.ITcoTaskStatus
ClearUserData := THIS^._clearUserDataTask.Invoke();
END_METHOD

(*~
	<docu>
		<summary>
			Gets the `ClearUserDataTask` task that controls clearing of the user data. 		
		</summary>			
	</docu>	
~*)
PROPERTY ClearUserDataTask : TcoCore.ITcoTaskStatus
GET
ClearUserDataTask := THIS^._clearUserDataTask;
END_GET
END_PROPERTY

(*~
	<docu>
		<summary>
			Gets the configuration of the sensor. 					
		</summary>			
	</docu>	
~*)
PROPERTY Config : REFERENCE TO TcoInsightConfig_v_5_x_x
GET
Config REF= _config;
END_GET
END_PROPERTY

METHOD FB_init : BOOL
VAR_INPUT
	bInitRetains : BOOL; // if TRUE, the retain variables are initialized (warm start / cold start)
	bInCopyCode : BOOL;  // if TRUE, the instance afterwards gets moved into the copy code (online change)
	ParentObject : ITcoObject;
END_VAR
END_METHOD

METHOD GetResultAsByte : BYTE
VAR_INPUT
    inPosition : UINT;
END_VAR
VAR
	_size : UINT;
END_VAR
_size := SIZEOF(GetResultAsByte);

IF (inPosition +_size) > THIS^._config.ResultDataSize THEN
	Messenger.Warning('<#Index of the ResultData in the method GetResultAsByte exceeds the size hardware structure mapped!#>');
	RETURN;
END_IF

IF (inPosition +_size) > TcoVisionParams.MAX_BYTE_ARRAY THEN
	Messenger.Programming('<#Index of the ResultData in the method GetResultAsByte exceeds the defined size!#>');
	RETURN;
END_IF

GetResultAsByte := THIS^._results.InspectionResults[inPosition];
END_METHOD

METHOD GetResultAsDint : DINT
VAR_INPUT
    inPosition : UINT;
END_VAR
VAR
	_index : UINT;
	_size : UINT;
END_VAR
_size := SIZEOF(GetResultAsDint);

IF (inPosition +_size) > THIS^._config.ResultDataSize THEN
	Messenger.Warning('<#Index of the ResultData in the method GetResultAsDint exceeds the size hardware structure mapped!#>');
	RETURN;
END_IF

IF (inPosition +_size) > TcoVisionParams.MAX_BYTE_ARRAY THEN
	Messenger.Programming('<#Index of the ResultData in the method GetResultAsDint exceeds the defined size!#>');
	RETURN;
END_IF

GetResultAsDint := TcoUtilities.TcoBytesToDint(THIS^._config.DataFormat,	THIS^._results.InspectionResults[inPosition],
															THIS^._results.InspectionResults[inPosition+1],
															THIS^._results.InspectionResults[inPosition+2],
															THIS^._results.InspectionResults[inPosition+3]);
END_METHOD

METHOD GetResultAsReal : REAL
VAR_INPUT
    inPosition : UINT;
END_VAR
VAR
	_index : UINT;
	_size : UINT;
END_VAR
_size := SIZEOF(GetResultAsReal);

IF (inPosition +_size) > THIS^._config.ResultDataSize THEN
	Messenger.Warning('<#Index of the ResultData in the method GetResultAsReal exceeds the size hardware structure mapped!#>');
	RETURN;
END_IF

IF (inPosition +_size) > TcoVisionParams.MAX_BYTE_ARRAY THEN
	Messenger.Programming('<#Index of the ResultData in the method GetResultAsReal exceeds the defined size!#>');
	RETURN;
END_IF

GetResultAsReal := TcoUtilities.TcoBytesToReal(THIS^._config.DataFormat,	THIS^._results.InspectionResults[inPosition],
															THIS^._results.InspectionResults[inPosition+1],
															THIS^._results.InspectionResults[inPosition+2],
															THIS^._results.InspectionResults[inPosition+3]);
END_METHOD

METHOD GetResultAsString : STRING
VAR_INPUT
    inPosition : UINT;
	inLength : UINT;
END_VAR
VAR
	_index : UINT;
	_bufferSize : UINT; 
	_resultString : STRING;
END_VAR

IF (inPosition +inLength) > THIS^._config.ResultDataSize THEN
	Messenger.Warning('<#Index of the ResultData in the method GetResultAsString exceeds the size hardware structure mapped!#>');
	RETURN;
END_IF

IF (inPosition +inLength) > TcoVisionParams.MAX_BYTE_ARRAY THEN
	Messenger.Programming('<#Index of the ResultData in the method GetResultAsString exceeds the defined size!#>');
	RETURN;
END_IF

_resultString:='';

IF (inLength>0) THEN 
	FOR	_index := 0 TO inLength-1 BY 1 DO	
		IF(THIS^._results.InspectionResults[inPosition + _index] <> 0) THEN
			_resultString := CONCAT(_resultString, F_ToCHR(THIS^._results.InspectionResults[inPosition + _index]));
		ELSE
			EXIT;	
		END_IF		
	END_FOR;
END_IF

GetResultAsString := _resultString;
END_METHOD

(*~
	<docu>
		<summary>
			Changes the job by its name. 		
		</summary>			
	</docu>	
~*)
METHOD ChangeJobByName : TcoCore.ITcoTaskStatus
VAR_INPUT
	inJobName : STRING;
END_VAR
ChangeJobByName := THIS^._changeJobByNameTask.InvokeWithParameters(inJobName);
END_METHOD

(*~
	<docu>
		<summary>
			Gets the `ClearResultDataTask` task that controls clearing of the results data. 		
		</summary>			
	</docu>	
~*)
PROPERTY ChangeJobByNameTask : TcoCore.ITcoTaskStatus
GET
ChangeJobByNameTask := THIS^._changeJobByNameTask;
END_GET
END_PROPERTY

(*~
	<docu>
		<summary>
			Changes the job by its identification number. 		
		</summary>			
	</docu>	
~*)
METHOD ChangeJobByNumber : TcoCore.ITcoTaskStatus
VAR_INPUT
	inJobNumber : UINT;
END_VAR
ChangeJobByNumber := THIS^._changeJobByNumberTask.InvokeWithParameters(inJobNumber);
END_METHOD

(*~
	<docu>
		<summary>
			Gets the `ClearResultDataTask` task that controls clearing of the results data. 		
		</summary>			
	</docu>	
~*)
PROPERTY ChangeJobByNumberTask : TcoCore.ITcoTaskStatus
GET
ChangeJobByNumberTask := THIS^._changeJobByNumberTask;
END_GET
END_PROPERTY

METHOD INTERNAL CheckIfOnline
VAR_INST
	_onlineTimer : TON;
END_VAR

IF NOT THIS^.inoIoData.AcquisitionStatus.Online THEN
	THIS^._status.CurrentJobName := '';
	THIS^._status.CurrentJobNumber := -1;
END_IF

_onlineTimer(IN:=NOT THIS^.inoIoData.AcquisitionControl.SetOffline AND NOT THIS^.inoIoData.AcquisitionStatus.Online,PT:=T#3S);

